# B&R Automation Studio project KeePak_BlissNewScreen
Automation Studio 4.7.5.60 SP

## Configuration MasterConfiguration_ServoRam

### Acp10map.ncm - X20CP0484/Motion/Acp10map.ncm
```
NcMapping (NcSwId=Acp10, DisabledNodesAreHidden=False)
  NcObject 8EI2X2HWT10.xxxx-1a_ncV_AXIS1 (ModuleId=8EI2X2HWT10.xxxx-1a, Type=ncV_AXIS, Channel=1, Disabled=TRUE, ModuleDisabled=FALSE)
  NcObject gServoRam (ModuleId=8EI2X2HWT10.xxxx-1a, Type=ncAXIS, Channel=1, AcoposSimulation=Off, InitParameter=gFeedi, AcoposParameter=brake, Disabled=FALSE, ModuleDisabled=FALSE)
  NcObject 8EI2X2HWT10.xxxx-1_ncV_AXIS1 (ModuleId=8EI2X2HWT10.xxxx-1, Type=ncV_AXIS, Channel=1, Disabled=TRUE, ModuleDisabled=FALSE)
  NcObject gBodyHopper (ModuleId=8EI2X2HWT10.xxxx-1, Type=ncAXIS, Channel=1, AcoposSimulation=Off, InitParameter=gFeedi, AcoposParameter=gBHop, Disabled=FALSE, ModuleDisabled=FALSE)
  NcObject 8EI2X2HWT10.xxxx-1a_ncV_AXIS2 (ModuleId=8EI2X2HWT10.xxxx-1a, Type=ncV_AXIS, Channel=2, Disabled=TRUE, ModuleDisabled=FALSE)
  NcObject gServoPnP (ModuleId=8EI2X2HWT10.xxxx-1a, Type=ncAXIS, Channel=2, AcoposSimulation=Off, InitParameter=gFeedi, AcoposParameter=disablebra, Disabled=FALSE, ModuleDisabled=FALSE)
  NcObject 8EI2X2HWT10.xxxx-1_ncV_AXIS2 (ModuleId=8EI2X2HWT10.xxxx-1, Type=ncV_AXIS, Channel=2, Disabled=TRUE, ModuleDisabled=FALSE)
  NcObject gLeftHopper (ModuleId=8EI2X2HWT10.xxxx-1, Type=ncAXIS, Channel=2, AcoposSimulation=Off, InitParameter=gFeedi, AcoposParameter=gBHop, Disabled=FALSE, ModuleDisabled=FALSE)
  NcObject 8EI2X2HWT10.xxxx-1a_ncV_AXIS3 (ModuleId=8EI2X2HWT10.xxxx-1a, Type=ncV_AXIS, Channel=3, Disabled=TRUE, ModuleDisabled=FALSE)
  NcObject gServoFeed (ModuleId=8EI2X2HWT10.xxxx-1a, Type=ncAXIS, Channel=3, AcoposSimulation=Off, InitParameter=gFeedi, AcoposParameter=disablebra, Disabled=FALSE, ModuleDisabled=FALSE)
  NcObject 8EI2X2HWT10.xxxx-1_ncV_AXIS3 (ModuleId=8EI2X2HWT10.xxxx-1, Type=ncV_AXIS, Channel=3, Disabled=TRUE, ModuleDisabled=FALSE)
  NcObject gRightHopper (ModuleId=8EI2X2HWT10.xxxx-1, Type=ncAXIS, Channel=3, AcoposSimulation=Off, InitParameter=gFeedi, AcoposParameter=gBHop, Disabled=FALSE, ModuleDisabled=FALSE)
```

### BodyHop.mpaxisbasic - X20CP0484/Motion/BodyHop.mpaxisbasic
```
Element mpBodyHopper (Type=mpaxisbasic)
  AxisConfiguration:
    Axis:
      MeasurementUnit = 1
  Alarms = MpAlarmX
    mapp.AlarmX.Core.Configuration:
      [0]:
        Severity = 110
      [1]:
        Severity = 110
      [2]:
        Severity = 110
      [3]:
        Severity = 110
      [4]:
        Severity = 110
      [5]:
        Severity = 110
      [6]:
        Severity = 110
      [7]:
        Severity = 110
      [8]:
        Severity = 110
      [9]:
        Severity = 110
      [10]:
        Severity = 110
      [11]:
        Severity = 110
      [12]:
        Severity = 110
      [13]:
        Severity = 110
      [14]:
        Severity = 110
      [15]:
        Severity = 110
```

### ServoPnP.mpaxisbasic - X20CP0484/Motion/ServoPnP.mpaxisbasic
```
Element mpServoPick (Type=mpaxisbasic)
  AxisConfiguration:
    Axis:
      MeasurementUnit = 1
  Alarms = MpAlarmX
    mapp.AlarmX.Core.Configuration:
      [0]:
        Severity = 110
      [1]:
        Severity = 110
      [2]:
        Severity = 110
      [3]:
        Severity = 110
      [4]:
        Severity = 110
      [5]:
        Severity = 110
      [6]:
        Severity = 110
      [7]:
        Severity = 110
      [8]:
        Severity = 110
      [9]:
        Severity = 110
      [10]:
        Severity = 110
      [11]:
        Severity = 110
      [12]:
        Severity = 110
      [13]:
        Severity = 110
      [14]:
        Severity = 110
      [15]:
        Severity = 110
```

- Safety project (password-protected, skipped)

## Logical view

### Global.var
```iecst
VAR
	GuideCylinder : BOOL;
	gForceBodyKicker : BOOL;
END_VAR
VAR RETAIN
	BodyHopperFirstHomeExecuted : BOOL;
	BodyHopper_EPD : MC_ENDLESS_POSITION;
END_VAR
VAR
	b_ModuleStatus : BOOL;
END_VAR
VAR RETAIN
	CycleCount : UDINT;
END_VAR
VAR
	DistanceAfterLatch : REAL;
	FeedInCycle : BOOL;
	FeedPosFinal : LREAL;
	FeedPositionCapture : LREAL;
	FeedServoBusy : BOOL;
	gActivePage : USINT;
	gAdhesiveCtrlInterface : AdhesiveCtrlInterface_typ;
	gAirPressureAlarmActive : BOOL;
	gAlarmActive : BOOL;
	gAlarmSystemActive : BOOL;
	gAutoTune : BOOL;
	gBodyHopper : ACP10AXIS_typ;
	gBodyHopperInterface : Axis_Interface_typ;
	gBotLinAxis : ACP10AXIS_typ;
	gBotLinAxis_1 : ACP10AXIS_typ;
	gChangePage : USINT;
	gCurrentLimitHit : BOOL;
	gCyclesToFinish : SINT;
	gDownstreamBlocked : BOOL;
END_VAR
VAR RETAIN
	gEndlessPosBot : MC_ENDLESS_POSITION;
	gEndlessPosTop : MC_ENDLESS_POSITION;
END_VAR
VAR
	gFoldPushCtrlInterface : FoldPushCtrlInterface_typ := (Parameters:=(LinMotBotFolder:=(Parameter:=(MpBasicParameters:=(Home:=(Mode:=mpAXIS_HOME_MODE_RESTORE_POS,Position:=0,StartVelocity:=25,HomingVelocity:=5,Acceleration:=500,StartDirection:=mpAXIS_HOME_DIR_NEGATIVE,TorqueLimit:=0.5,BlockDetectionPositionError:=4,PositionErrorStopLimit:=10),Jog:=(Velocity:=2)))),LinMotTopFolder:=(Parameter:=(MpBasicParameters:=(Home:=(Mode:=mpAXIS_HOME_MODE_RESTORE_POS,Position:=0,StartVelocity:=25,HomingVelocity:=5,Acceleration:=500,StartDirection:=mpAXIS_HOME_DIR_NEGATIVE,TorqueLimit:=0.5,BlockDetectionPositionError:=4,PositionErrorStopLimit:=10),Jog:=(Velocity:=2))))));
	gHighSeverityAlarmActive : BOOL;
	gHMI : HMIControl_typ;
	gHomingParameters : Home_Parameters_typ;
	gIO : IO_typ;
	gIsSimulated : BOOL;
	gLeftHopper : ACP10AXIS_typ;
	gLeftHopperInterface : Axis_Interface_typ;
	gLowSeverityAlarmActive : BOOL;
	gModeControlInterface : ModeCtrlInterface_typ;
	gNumActiveAlarms : UDINT;
	gNumAlarms : UDINT;
	gOffDelayCompensation : REAL;
	gOnDelayCompensation : REAL;
	gPassword : ARRAY[0..2] OF STRING[80] := ['','1111','2147'];
	gPnPAtStopPosition : BOOL;
	gPusherOn : BOOL;
	gRamAtStopPosition : BOOL;
	gRamCtrlInterface : RamControlInterface_typ;
	gRamWaitingOnBox : BOOL;
END_VAR
VAR RETAIN
	gRecipeInterface : {REDUND_UNREPLICABLE} RecipeCtrlInterface_typ := (0);
END_VAR
VAR
	gRightHopper : ACP10AXIS_typ;
	gRightHopperInterface : Axis_Interface_typ;
	gSafetyNotOKAlarmActive : BOOL;
	gServoFeed : ACP10AXIS_typ;
	gServoFeedInterface : Axis_Interface_typ;
	gServoFeed_1 : ACP10AXIS_typ;
	gServoPnP : ACP10AXIS_typ;
	gServoPnPInterface : Axis_Interface_typ;
	gServoRam : ACP10AXIS_typ;
	gServoRamInterface : Axis_Interface_typ;
	gServoRam_1 : ACP10AXIS_typ;
	gSoftwareReset : BOOL;
	gTopLinAxis : ACP10AXIS_typ;
	gTopLinAxis_1 : ACP10AXIS_typ;
	gUserLevel : USINT;
	gVacCtrlInterface : VacCtrlInterface_typ;
	HoperLowStop : BOOL;
	HopperLowTime : TIME := T#7s;
	InfeedBoxPresent : BOOL;
END_VAR
VAR RETAIN
	LeftHopperFirstHomeExecuted : BOOL;
	LeftHopper_EPD : MC_ENDLESS_POSITION;
	LubeCount : UDINT;
END_VAR
VAR
	LubricationOK : BOOL;
	Melter : DUT_NDSN_Flex;
	PhotoEyeSeen : BOOL;
END_VAR
VAR RETAIN
	RightHopperFirstHomeExecuted : BOOL;
	RightHopper_EPD : MC_ENDLESS_POSITION;
	ServoFeedFirstHomeExecuted : BOOL;
	ServoFeed_EPD : MC_ENDLESS_POSITION;
END_VAR
VAR
	ServoPnPAutoHome : BOOL;
END_VAR
VAR RETAIN
	ServoPnPFirstHomeExecuted : BOOL;
	ServoPnP_EPD : MC_ENDLESS_POSITION;
END_VAR
VAR
	ServoRamAutoHome : BOOL;
	ServoRamBusy : BOOL;
	ServoRamClear : BOOL;
END_VAR
VAR RETAIN
	ServoRamFirstHomeExecuted : BOOL;
END_VAR
VAR
	ServoRamTrigger : BOOL;
END_VAR
VAR RETAIN
	ServoRam_EPD : MC_ENDLESS_POSITION;
END_VAR
VAR
	StopFeed : BOOL;
END_VAR
```

### Program Logical/Actuators/NordsonComm/NordsonMBComm

#### MbApp.st
```iecst
(********************************************************************
 * COPYRIGHT -- Bernecker + Rainer
 ********************************************************************
 * Program: MbApp
 * File: MbApp.st
 * Author: Bernecker + Rainer
 * Created: October 22, 2009
 ********************************************************************
 * Implementation of program MbApp
 * State Nomenclature: "request" is a write to the nordson melter asking for some data
 * 					   "read" is a read from the nordson melter of the previously requested data
 *                     "write" is a write to the nordson melter asking to write some data to the melter
 *                     "verify" is a read from the nordson melter where we check to see that the write was accepted
 ********************************************************************)

PROGRAM _INIT

	NordsonTxPacket.Byte0_MelterControl := 16#1;
	NordsonTxPacket.Byte1_Command := 3;
	NordsonTxPacket.Byte2_Data_Index := 16#78;
	NordsonTxPacket.Byte3_Channel_Num := 16#3;
	NordsonTxPacket.Byte4_5_WriteData := 0;
	NordsonTxPacket.Byte6_7_Mot1Spd := 0;
	NordsonTxPacket.Byte8_9_Mot2Spd := 0;
	NordsonTxPacket.Byte10_11_Mot3Spd := 0;
	NordsonTxPacket.Byte12_13_Mot4Spd := 0;
	NordsonTxPacket.Byte14_15_NotUsed := 0;

	state := MB_IDLE;

	(* init values *)
	mb_station 			:= 'IF2.ST2';					(* path to modbus station *)
	write_register_address	:= 1024;						(* register address on modbus station *)
	read_register_address	:= 0;						(* register address on modbus station *)
	num_registers_to_write := 8;
	num_registers_to_read := 8;

	testChannel := CHANNEL_ACT_TEMP_START;
	testIdx := IDX_ACT_TEMP;

	gAdhesiveCtrlInterface.Commands.MelterOn := TRUE;
	gAdhesiveCtrlInterface.Commands.PumpsOn := TRUE;
	//gAdhesiveCtrlInterface.Parameters.NordsonComms.StandbyTimeoutTime := T#2h;
	//Removed Standby due to Waco machine going into Standby at random times. Added 05/15/2024

	FirstTimeCopySetTemps := FALSE;

END_PROGRAM

PROGRAM _CYCLIC

	IF(gAdhesiveCtrlInterface.Parameters.FeedbackIsModbusTCP) THEN
		gHMI.StatusDatapoints.NordsonModbusSDP := UNHIDE + UNLOCK;
	ELSE
		gHMI.StatusDatapoints.NordsonModbusSDP := HIDE + LOCK;
	END_IF

	StandbyTimer.IN := NOT(gRamCtrlInterface.Status.Running) AND NOT(gAdhesiveCtrlInterface.Commands.MelterStandbyOn);
	StandbyTimer.PT := gAdhesiveCtrlInterface.Parameters.NordsonComms.StandbyTimeoutTime;
	StandbyTimer();

	IF(StandbyTimer.Q) THEN
		gAdhesiveCtrlInterface.Commands.MelterStandbyOn := TRUE;
	END_IF

	//clearing standby on command shiuld turn standby off. Changed standbyoff to True
	IF(gAdhesiveCtrlInterface.Commands.MelterStandbyOff) THEN
		gAdhesiveCtrlInterface.Commands.MelterStandbyOff := TRUE;
		gAdhesiveCtrlInterface.Commands.MelterStandbyOn := FALSE;
	END_IF

	IF((gAdhesiveCtrlInterface.Status.NordsonInStandby) AND (gAdhesiveCtrlInterface.Parameters.FeedbackIsModbusTCP)) THEN
		gHMI.StatusDatapoints.NordsonStandbyOffSDP := UNHIDE + UNLOCK;
	ELSE
		gHMI.StatusDatapoints.NordsonStandbyOffSDP := HIDE + LOCK;
	END_IF

	//if nordson feedback is bypassed, the error count should reset to 0
	IF gAdhesiveCtrlInterface.Parameters.NordsonComms.ByPassFeedback THEN
		gAdhesiveCtrlInterface.Parameters.NordsonComms.ConsecutiveErrorCount := 0;
	END_IF

	CASE state OF

		MB_IDLE:
			FeedbackCycleTimer.IN := ((gAdhesiveCtrlInterface.Parameters.FeedbackIsModbusTCP) AND (gAdhesiveCtrlInterface.Parameters.NordsonComms.ByPassFeedback = FALSE));

			IF(gAdhesiveCtrlInterface.Parameters.FeedbackIsModbusTCP = FALSE) THEN
				gAdhesiveCtrlInterface.Parameters.NordsonComms.ConsecutiveErrorCount := 0;
			END_IF

			IF(gAdhesiveCtrlInterface.Commands.WriteChannelTemp) THEN
				gAdhesiveCtrlInterface.Commands.WriteChannelTemp := FALSE;
				TempChannelToWrite := 0;
				state := MB_WRITE_SET_TEMP;

			ELSIF(FeedbackCycleTimer.Q) THEN
				FeedbackCycleTimer.IN := FALSE;
				state := MB_REQUEST_MELTER_STATUS;
			END_IF

		MB_REQUEST_MELTER_STATUS:

			WriteMultipleRegisters.enable := 1;
			NordsonTxPacket.Byte0_MelterControl := MelterCmd;
			NordsonTxPacket.Byte1_Command := READ_COMMAND;
			NordsonTxPacket.Byte2_Data_Index := IDX_MELTER_STATUS;
			NordsonTxPacket.Byte3_Channel_Num := 0;

			IF((WriteMultipleRegisters.status = ERR_FUB_ENABLE_FALSE) OR (WriteMultipleRegisters.status = ERR_FUB_BUSY)) THEN
				//do nothing
			ELSIF(WriteMultipleRegisters.status = ERR_OK) THEN
				WriteMultipleRegisters.enable := 0;
				state := MB_READ_MELTER_STATUS;
			ELSE
				WriteMultipleRegisters.enable := 0;
				MBError := WriteMultipleRegisters.status;
				state := MB_ERROR;
			END_IF

		MB_READ_MELTER_STATUS:

			ReadMultipleRegisters.enable := 1;

			IF((ReadMultipleRegisters.status = ERR_FUB_ENABLE_FALSE) OR (ReadMultipleRegisters.status = ERR_FUB_BUSY)) THEN
				//do nothing
			ELSIF(ReadMultipleRegisters.status = ERR_OK) THEN

				ReadMultipleRegisters.enable := 0;

				IF(NordsonRxPacket.Byte2_Ack_Data_Index = NordsonTxPacket.Byte2_Data_Index) THEN

					gAdhesiveCtrlInterface.Parameters.NordsonComms.MelterStatus := NordsonRxPacket.Byte4_5_Read_Data_0;
					gAdhesiveCtrlInterface.Parameters.NordsonComms.MelterIsOn := (gAdhesiveCtrlInterface.Parameters.NordsonComms.MelterStatus <> 8); //melter status == 8 => melter is not on

					DecodeStatus;

					//the melter MUST see a 0 for its ON command before it sees a 1. Send a 0 if the unit is faulted OR we have previously told it to turn on. and it never came on
				//	IF((gAdhesiveCtrlInterface.Parameters.NordsonComms.UnitFaulted) OR ((gAdhesiveCtrlInterface.Parameters.NordsonComms.MelterIsOn = FALSE) AND (NordsonTxPacket.Byte0_MelterControl.0 = TRUE))) THEN
					IF((gAdhesiveCtrlInterface.Parameters.NordsonComms.MelterIsOn = FALSE) AND (NordsonTxPacket.Byte0_MelterControl.0 = TRUE)) THEN
						MelterCmd := MELTER_OFF + PUMPS_OFF; //melter off, pumps off
					ELSE

						MelterCmd := 0;
						IF(gAdhesiveCtrlInterface.Commands.MelterOn) THEN
							MelterCmd := MelterCmd + MELTER_ON;
						END_IF

						IF((gAdhesiveCtrlInterface.Commands.PumpsOn) AND (gAdhesiveCtrlInterface.Status.UnitReady)) THEN
							MelterCmd := MelterCmd + PUMPS_ON; //only turn the pump on if the melter is ready
						END_IF

						IF((gAdhesiveCtrlInterface.Commands.MelterStandbyOn = FALSE) OR ((gAdhesiveCtrlInterface.Status.NordsonInStandby = FALSE) AND NordsonTxPacket.Byte0_MelterControl.6 = TRUE)) THEN
							//do not standby on
						ELSIF (gAdhesiveCtrlInterface.Commands.MelterStandbyOn = TRUE) THEN
							MelterCmd := MelterCmd + STANDBY_ON; //only turn the pump on if the melter is ready
						END_IF
					END_IF

					state := MB_REQUEST_SET_TEMPS;
				ELSE
					//stay in this state and re-execute read
				END_IF

			ELSE
				ReadMultipleRegisters.enable := 0;
				MBError := ReadMultipleRegisters.status;
				state := MB_ERROR;
			END_IF

		MB_REQUEST_SET_TEMPS:

			WriteMultipleRegisters.enable := 1;
			NordsonTxPacket.Byte0_MelterControl := MelterCmd;
			NordsonTxPacket.Byte1_Command := READ_COMMAND;
			NordsonTxPacket.Byte2_Data_Index := IDX_SET_TEMP;
			NordsonTxPacket.Byte3_Channel_Num := CHANNEL_SET_TEMP_START;

			IF((WriteMultipleRegisters.status = ERR_FUB_ENABLE_FALSE) OR (WriteMultipleRegisters.status = ERR_FUB_BUSY)) THEN
				//do nothing
			ELSIF(WriteMultipleRegisters.status = ERR_OK) THEN
				WriteMultipleRegisters.enable := 0;
				gAdhesiveCtrlInterface.Parameters.NordsonComms.ConsecutiveErrorCount := 0;
				state := MB_READ_SET_TEMPS;
			ELSE
				WriteMultipleRegisters.enable := 0;
				MBError := WriteMultipleRegisters.status;
				state := MB_ERROR;
			END_IF

		MB_READ_SET_TEMPS:

			ReadMultipleRegisters.enable := 1;

			IF((ReadMultipleRegisters.status = ERR_FUB_ENABLE_FALSE) OR (ReadMultipleRegisters.status = ERR_FUB_BUSY)) THEN
				//do nothing
			ELSIF(ReadMultipleRegisters.status = ERR_OK) THEN
				ReadMultipleRegisters.enable := 0;
				gAdhesiveCtrlInterface.Parameters.NordsonComms.ConsecutiveErrorCount := 0;

				IF((NordsonRxPacket.Byte2_Ack_Data_Index = NordsonTxPacket.Byte2_Data_Index) AND
					(NordsonRxPacket.Byte3_Ack_Channel_Num = NordsonTxPacket.Byte3_Channel_Num)) THEN

					DecodeStatus;

					gAdhesiveCtrlInterface.Parameters.NordsonComms.ChannelSetTempActual[0] := NordsonRxPacket.Byte4_5_Read_Data_0;
					gAdhesiveCtrlInterface.Parameters.NordsonComms.ChannelSetTempActual[1] := NordsonRxPacket.Byte6_7_Read_Data_1;
					gAdhesiveCtrlInterface.Parameters.NordsonComms.ChannelSetTempActual[2] := NordsonRxPacket.Byte8_9_Read_Data_2;
					gAdhesiveCtrlInterface.Parameters.NordsonComms.ChannelSetTempActual[3] := NordsonRxPacket.Byte10_11_Read_Data_3;
					gAdhesiveCtrlInterface.Parameters.NordsonComms.ChannelSetTempActual[4] := NordsonRxPacket.Byte12_13_Read_Data_4;
                    gAdhesiveCtrlInterface.Parameters.NordsonComms.ChannelSetTempActual[5] := NordsonRxPacket.Byte14_15_Read_Data_5;
//                    gAdhesiveCtrlInterface.Parameters.NordsonComms.ChannelSetTempActual[6] := NordsonRxPacket.Byte16_17_Read_Data_6;
//                    gAdhesiveCtrlInterface.Parameters.NordsonComms.ChannelSetTempActual[7] := NordsonRxPacket.Byte18_19_Read_Data_7;

                    IF (FirstTimeCopySetTemps = FALSE) THEN
						gAdhesiveCtrlInterface.Parameters.NordsonComms.ChannelSetTempRequested := gAdhesiveCtrlInterface.Parameters.NordsonComms.ChannelSetTempActual;
						FirstTimeCopySetTemps := TRUE;
					END_IF

					state := MB_REQUEST_ACT_TEMPS; //for now, just go back to idle. Future versions need to read more stuff
				ELSE
					//stay in this state and re-execute read
				END_IF
			ELSE
				ReadMultipleRegisters.enable := 0;
				MBError := ReadMultipleRegisters.status;
				state := MB_ERROR;
			END_IF

		MB_REQUEST_ACT_TEMPS:

			WriteMultipleRegisters.enable := 1;
			NordsonTxPacket.Byte0_MelterControl := MelterCmd;
			NordsonTxPacket.Byte1_Command := READ_COMMAND;
			NordsonTxPacket.Byte2_Data_Index := IDX_ACT_TEMP;
			NordsonTxPacket.Byte3_Channel_Num := CHANNEL_ACT_TEMP_START;

			IF((WriteMultipleRegisters.status = ERR_FUB_ENABLE_FALSE) OR (WriteMultipleRegisters.status = ERR_FUB_BUSY)) THEN
				//do nothing
			ELSIF(WriteMultipleRegisters.status = ERR_OK) THEN
				WriteMultipleRegisters.enable := 0;
				state := MB_READ_ACT_TEMPS;
			ELSE
				WriteMultipleRegisters.enable := 0;
				MBError := WriteMultipleRegisters.status;
				state := MB_ERROR;
			END_IF

		MB_READ_ACT_TEMPS:

			ReadMultipleRegisters.enable := 1;

			IF((ReadMultipleRegisters.status = ERR_FUB_ENABLE_FALSE) OR (ReadMultipleRegisters.status = ERR_FUB_BUSY)) THEN
				//do nothing
			ELSIF(ReadMultipleRegisters.status = ERR_OK) THEN
				ReadMultipleRegisters.enable := 0;

				IF((NordsonRxPacket.Byte2_Ack_Data_Index = NordsonTxPacket.Byte2_Data_Index) AND
					(NordsonRxPacket.Byte3_Ack_Channel_Num = NordsonTxPacket.Byte3_Channel_Num)) THEN

					DecodeStatus;

					gAdhesiveCtrlInterface.Parameters.NordsonComms.ChannelActTemp[0] := NordsonRxPacket.Byte4_5_Read_Data_0;
					gAdhesiveCtrlInterface.Parameters.NordsonComms.ChannelActTemp[1] := NordsonRxPacket.Byte6_7_Read_Data_1;
					gAdhesiveCtrlInterface.Parameters.NordsonComms.ChannelActTemp[2] := NordsonRxPacket.Byte8_9_Read_Data_2;
					gAdhesiveCtrlInterface.Parameters.NordsonComms.ChannelActTemp[3] := NordsonRxPacket.Byte10_11_Read_Data_3;
					gAdhesiveCtrlInterface.Parameters.NordsonComms.ChannelActTemp[4] := NordsonRxPacket.Byte12_13_Read_Data_4;
                    gAdhesiveCtrlInterface.Parameters.NordsonComms.ChannelActTemp[5] := NordsonRxPacket.Byte14_15_Read_Data_5;
//                    gAdhesiveCtrlInterface.Parameters.NordsonComms.ChannelActTemp[6] := NordsonRxPacket.Byte16_17_Read_Data_6;
//                    gAdhesiveCtrlInterface.Parameters.NordsonComms.ChannelActTemp[7] := NordsonRxPacket.Byte18_19_Read_Data_7;
//                    gAdhesiveCtrlInterface.Parameters.NordsonComms.ChannelActTemp[8] := NordsonRxPacket.Byte20_21_Read_Data_8;
//                    gAdhesiveCtrlInterface.Parameters.NordsonComms.ChannelActTemp[9] := NordsonRxPacket.Byte22_23_Read_Data_9;
//                    gAdhesiveCtrlInterface.Parameters.NordsonComms.ChannelActTemp[10] := NordsonRxPacket.Byte24_25_Read_Data_10;

					state := MB_REQUEST_ATS_ALARMS;
				ELSE
					//stay in this state and re-execute read
				END_IF

			ELSE
				ReadMultipleRegisters.enable := 0;
				MBError := ReadMultipleRegisters.status;
				state := MB_ERROR;
			END_IF

		MB_REQUEST_ATS_ALARMS:

			WriteMultipleRegisters.enable := 1;
			NordsonTxPacket.Byte0_MelterControl := MelterCmd;
			NordsonTxPacket.Byte1_Command := READ_COMMAND;
			NordsonTxPacket.Byte2_Data_Index := IDX_ATS_ALARMS;

			IF((WriteMultipleRegisters.status = ERR_FUB_ENABLE_FALSE) OR (WriteMultipleRegisters.status = ERR_FUB_BUSY)) THEN
				//do nothing
			ELSIF(WriteMultipleRegisters.status = ERR_OK) THEN
				WriteMultipleRegisters.enable := 0;
				state := MB_READ_ATS_ALARMS;
			ELSE
				WriteMultipleRegisters.enable := 0;
				MBError := WriteMultipleRegisters.status;
				state := MB_ERROR;
			END_IF

		MB_READ_ATS_ALARMS:

			ReadMultipleRegisters.enable := 1;

			IF((ReadMultipleRegisters.status = ERR_FUB_ENABLE_FALSE) OR (ReadMultipleRegisters.status = ERR_FUB_BUSY)) THEN
				//do nothing
			ELSIF(ReadMultipleRegisters.status = ERR_OK) THEN
				ReadMultipleRegisters.enable := 0;

				IF(NordsonRxPacket.Byte2_Ack_Data_Index = NordsonTxPacket.Byte2_Data_Index) THEN

					DecodeStatus;

					gAdhesiveCtrlInterface.Status.ATS_AddOnOverLimit := NordsonRxPacket.Byte4_5_Read_Data_0.0;
					gAdhesiveCtrlInterface.Status.ATS_AddOnUnderLimit := NordsonRxPacket.Byte4_5_Read_Data_0.1;

					state := MB_IDLE;
				ELSE
					//stay in this state and re-execute read
				END_IF

			ELSE
				ReadMultipleRegisters.enable := 0;
				MBError := ReadMultipleRegisters.status;
				state := MB_ERROR;
			END_IF

		MB_WRITE_SET_TEMP:

			WriteMultipleRegisters.enable := 1;
			NordsonTxPacket.Byte0_MelterControl := MelterCmd;
			NordsonTxPacket.Byte1_Command := WRITE_COMMAND;
			NordsonTxPacket.Byte2_Data_Index := IDX_SET_TEMP;
			NordsonTxPacket.Byte3_Channel_Num := TempChannelToWrite + 1; //TempChannelToWrite starts counting at 0, but nordson melter starts counting at 1
			NordsonTxPacket.Byte4_5_WriteData := gAdhesiveCtrlInterface.Parameters.NordsonComms.ChannelSetTempRequested[TempChannelToWrite];

			IF((WriteMultipleRegisters.status = ERR_FUB_ENABLE_FALSE) OR (WriteMultipleRegisters.status = ERR_FUB_BUSY)) THEN
				//do nothing
			ELSIF(WriteMultipleRegisters.status = ERR_OK) THEN
				WriteMultipleRegisters.enable := 0;
				state := MB_VERIFY_SET_TEMP_WRITE;
			ELSE
				WriteMultipleRegisters.enable := 0;
				MBError := WriteMultipleRegisters.status;
				state := MB_ERROR;
			END_IF

		MB_VERIFY_SET_TEMP_WRITE:

			ReadMultipleRegisters.enable := 1;

			IF((ReadMultipleRegisters.status = ERR_FUB_ENABLE_FALSE) OR (ReadMultipleRegisters.status = ERR_FUB_BUSY)) THEN
				//do nothing
			ELSIF(ReadMultipleRegisters.status = ERR_OK) THEN
				ReadMultipleRegisters.enable := 0;

				IF((NordsonRxPacket.Byte2_Ack_Data_Index = NordsonTxPacket.Byte2_Data_Index) AND
					(NordsonRxPacket.Byte3_Ack_Channel_Num = NordsonTxPacket.Byte3_Channel_Num)) THEN

					DecodeStatus;

					IF(TempChannelToWrite < NUM_NORDSON_TEMP_ZONES_M1) THEN
						IF(TempChannelToWrite = 0) THEN
							TempChannelToWrite := 2; //channel 0 and 1 get the same temp, no need to re-write channel 1
							state := MB_WRITE_SET_TEMP;
						ELSE
							TempChannelToWrite := TempChannelToWrite + 1; //set the temperature for the next channel (Skip channel 2). Machine has 3 total channels
							state := MB_WRITE_SET_TEMP;
						END_IF
					ELSE
						state := MB_IDLE;
					END_IF
				ELSE
					//stay in this state and re-execute read
				END_IF

			ELSE
				ReadMultipleRegisters.enable := 0;
				MBError := ReadMultipleRegisters.status;
				state := MB_ERROR;
			END_IF

		MB_REQUEST_ADH_USE:

			WriteMultipleRegisters.enable := 1;
			NordsonTxPacket.Byte0_MelterControl := MelterCmd;
			NordsonTxPacket.Byte1_Command := READ_COMMAND;
			NordsonTxPacket.Byte2_Data_Index := IDX_ADHESIVE_HOUR;
			NordsonTxPacket.Byte3_Channel_Num := CHANNEL_ADHESIVE_HOUR;

			IF((WriteMultipleRegisters.status = ERR_FUB_ENABLE_FALSE) OR (WriteMultipleRegisters.status = ERR_FUB_BUSY)) THEN
				//do nothing
			ELSIF(WriteMultipleRegisters.status = ERR_OK) THEN
				WriteMultipleRegisters.enable := 0;
				state := MB_READ_ACT_TEMPS;
			ELSE
				WriteMultipleRegisters.enable := 0;
				MBError := WriteMultipleRegisters.status;
				state := MB_ERROR;
			END_IF

		MB_READ_ADH_USE:

			ReadMultipleRegisters.enable := 1;

			IF((ReadMultipleRegisters.status = ERR_FUB_ENABLE_FALSE) OR (ReadMultipleRegisters.status = ERR_FUB_BUSY)) THEN
				//do nothing
			ELSIF(ReadMultipleRegisters.status = ERR_OK) THEN
				ReadMultipleRegisters.enable := 0;

				IF((NordsonRxPacket.Byte2_Ack_Data_Index = NordsonTxPacket.Byte2_Data_Index) AND
					(NordsonRxPacket.Byte3_Ack_Channel_Num = NordsonTxPacket.Byte3_Channel_Num)) THEN

					//	NordsonData.AdhesiveUsePerHour := NordsonRxPacket.Byte4_5_Read_Data_0 + (NordsonRxPacket.Byte6_7_Read_Data_1*(65536)); //data 0 + data 1 shifted up 16 bits

					state := MB_READ_ACT_TEMPS;
				ELSE
					//stay in this state and re-execute read
				END_IF
			END_IF

		MB_WRITE_REGISTERS:

			WriteMultipleRegisters.enable := 1;
			NordsonTxPacket.Byte0_MelterControl := MELTER_ON;
			NordsonTxPacket.Byte1_Command := READ_COMMAND;
			NordsonTxPacket.Byte2_Data_Index := testChannel;
			NordsonTxPacket.Byte3_Channel_Num := testIdx;

			IF((WriteMultipleRegisters.status = ERR_FUB_ENABLE_FALSE) OR (WriteMultipleRegisters.status = ERR_FUB_BUSY)) THEN
				//do nothing
			ELSIF(WriteMultipleRegisters.status = ERR_OK) THEN
				WriteMultipleRegisters.enable := 0;
				state := MB_READ_ACT_TEMPS;
			ELSE
				WriteMultipleRegisters.enable := 0;
				MBError := WriteMultipleRegisters.status;
				state := MB_ERROR;
			END_IF

		MB_READ_REGISTERS:

			ReadMultipleRegisters.enable := 1;

			IF((ReadMultipleRegisters.status = ERR_FUB_ENABLE_FALSE) OR (ReadMultipleRegisters.status = ERR_FUB_BUSY)) THEN
				//do nothing
			ELSIF(ReadMultipleRegisters.status = ERR_OK) THEN
				ReadMultipleRegisters.enable := 0;
				state := MB_IDLE;
			ELSE
				ReadMultipleRegisters.enable := 0;
				MBError := ReadMultipleRegisters.status;
				state := MB_ERROR;
			END_IF

		MB_ERROR:
			gAdhesiveCtrlInterface.Parameters.NordsonComms.ConsecutiveErrorCount := gAdhesiveCtrlInterface.Parameters.NordsonComms.ConsecutiveErrorCount + 1;
		state := MB_IDLE; //keep re-trying indefinetly, logic below will set/reset alarms alarm

	END_CASE;

	IF EDGEPOS(gAdhesiveCtrlInterface.Parameters.NordsonComms.ConsecutiveErrorCount >= 10) THEN
		MpAlarmXSet(gAlarmXCore, ALARM_NORDSON_COMMS);
	ELSIF EDGENEG(gAdhesiveCtrlInterface.Parameters.NordsonComms.ConsecutiveErrorCount >= 10)THEN
		MpAlarmXReset(gAlarmXCore, ALARM_NORDSON_COMMS);
	END_IF

	IF EDGEPOS(gAdhesiveCtrlInterface.Status.ATS_AddOnOverLimit) THEN
		MpAlarmXSet(gAlarmXCore, ALARM_ATS_OVERLIMIT);
	ELSIF EDGENEG(gAdhesiveCtrlInterface.Status.ATS_AddOnOverLimit)THEN
		MpAlarmXReset(gAlarmXCore, ALARM_ATS_OVERLIMIT);
	END_IF

	IF EDGEPOS(gAdhesiveCtrlInterface.Status.ATS_AddOnUnderLimit) THEN
		MpAlarmXSet(gAlarmXCore, ALARM_ATS_UNDERLIMIT);
	ELSIF EDGENEG(gAdhesiveCtrlInterface.Status.ATS_AddOnUnderLimit)THEN
		MpAlarmXReset(gAlarmXCore, ALARM_ATS_UNDERLIMIT);
	END_IF

	IF EDGEPOS(gAdhesiveCtrlInterface.Status.NordsonInStandby) THEN
		MpAlarmXSet(gAlarmXCore, ALARM_NORDSON_STANDBY);
	ELSIF EDGENEG(gAdhesiveCtrlInterface.Status.NordsonInStandby)THEN
		MpAlarmXReset(gAlarmXCore, ALARM_NORDSON_STANDBY);
	END_IF

	//force unit ready and unit faulted status flags if ModbusTCP control is selected and bypass is enabled
	IF(gAdhesiveCtrlInterface.Parameters.FeedbackIsModbusTCP AND gAdhesiveCtrlInterface.Parameters.NordsonComms.ByPassFeedback) THEN
		gAdhesiveCtrlInterface.Parameters.NordsonComms.UnitReady := TRUE;
		gAdhesiveCtrlInterface.Parameters.NordsonComms.UnitFaulted := FALSE;
		gAdhesiveCtrlInterface.Status.ATS_AddOnOverLimit := FALSE;
		gAdhesiveCtrlInterface.Status.ATS_AddOnUnderLimit := FALSE;
	END_IF

	//Must be called after state machine. Do not move any function calls that are already below this line
	WriteMultipleRegisters.pStation := ADR(mb_station);
	WriteMultipleRegisters.startAddress := write_register_address;
	WriteMultipleRegisters.nrRegisters := num_registers_to_write;
	WriteMultipleRegisters.pData := ADR(NordsonTxPacket);
	WriteMultipleRegisters.dataSize := SIZEOF(NordsonTxPacket);
	WriteMultipleRegisters();

	ReadMultipleRegisters.pStation := ADR(mb_station);
	ReadMultipleRegisters.startAddress := read_register_address;
	ReadMultipleRegisters.nrRegisters := num_registers_to_read;
	ReadMultipleRegisters.pData := ADR(NordsonRxPacket);
	ReadMultipleRegisters.dataSize := SIZEOF(NordsonRxPacket);
	ReadMultipleRegisters();

	FeedbackCycleTimer.PT := gAdhesiveCtrlInterface.Parameters.NordsonComms.FeedbackTime;
	FeedbackCycleTimer();

				END_PROGRAM
```

### Program Logical/AsSafetySolution/SafetySample

#### SafetySample.st
```iecst
(********************************************************************
 * COPYRIGHT -- Bernecker + Rainer
 ********************************************************************
 * Program: SafetySample
 * File: SafetySample.st
 * Author: B&R
 ********************************************************************
 * Implementation of program SafetySample
 ********************************************************************)

PROGRAM _INIT

(*KEEPAK specific hard coded values *)
	remotecmd.Password 			:= 'safety';				(* password *)
	remotecmd.NewPassword	 	:= 'safety';				(* password *)
	appcmd1.Password 			:= 'safety';
	datacmd1.Password 			:= 'safety';
	datacmd2.Password 			:= 'safety';

	visuUsedSLIDRemote			:= 1;
	visuUsedSLIDData			:= 1;

	slxused						:= 1;
	Station						:= 'IF6.ST6';
	visuEnableMachineOptions	:= 1;
	visuEnableModuleFlags		:= 1;

	visuLockSDP					:= 2;

(* command structure for remote control FUB *)
remotecmd.Version := safeVERSION_R107;	(* version *)
//remotecmd.Password := '';				(* password *)

(* command structure for application download *)
appcmd1.Version := safeVERSION_R107;	(* version *)
//appcmd1.Password := '';					(* password *)
appcmd1.ApplicationID := 1;				(* application id *)

(* command structure for machine options download *)
datacmd1.Version := safeVERSION_R107;								(* version *)
//datacmd1.Password := '';											(* password *)
datacmd1.pDeviceListInput := ADR(visuDeviceListInput);				(* device list *)
datacmd1.pMachineOptionsInput := ADR(dataMachineOptionsBitInput);	(* bit machine options *)
datacmd1.pModuleFlagsInput := ADR(dataModuleFlagsInput);			(* module flags *)
datacmd1.pAcknMachineOptions := ADR(dataAcknMachineOptions);		(* acknowledge information *)

(* command structure for extended machine options *)
datacmd2.Version := safeVERSION_R107;					(* version *)
//datacmd2.Password := '';								(* password *)
datacmd2.pIntDataInput := ADR(visuIntInput);			(* INT channels *)
datacmd2.NumberIntInput := 1;							(* number of INT channels *)
datacmd2.pUintDataInput := ADR(visuUintInput);			(* UINT channels *)
datacmd2.NumberUintInput := 1;							(* number of UINT channels *)
datacmd2.pDintDataInput := ADR(visuDintInput);			(* DINT channels *)
datacmd2.NumberDintInput := 1;							(* number of DINT channels *)
datacmd2.pUdintDataInput := ADR(visuUdintInput);		(* UDINT channels *)
datacmd2.NumberUdintInput := 1;							(* number of UDINT channels *)
datacmd2.pAcknMachineOptions := ADR(visuAcknExtData);	(* acknowledge information *)

(* hide elements in visualization *)
FOR xcnt := 0 TO SIZEOF(statusButtonActiv) - 1 DO
	statusButtonActiv[xcnt] := 1;
END_FOR

(* hide elements in visualization *)
statusButtonUnlockApp := 1;
statusButtonUnlockData := 1;
statusAcknInfoData := 1;
statusButtonUnlockExtData := 1;
statusAcknInfoExtData := 1;
statusDialog := 1;

(* set SafeLOGIC ID *)
visuUsedSLIDRemote := 1;
visuUsedSLIDData := 1;

END_PROGRAM

PROGRAM _CYCLIC
	(****************************************************************************************************************************************)
	(****************************************************************************************************************************************)
	(****************************************************************************************************************************************)
	(* show dialog to ackn command *)
	IF (dialogRemoteCmd = 1) THEN
		statusDialog := 0;
		dialogRemoteCmd := 0;
		indexButtonLeft := 0;
		indexButtonRight := 1;
		indexHeaderText := 0;
		IF (remotecmd.Data = safeCMD_SK_FORMAT) THEN
			indexMessageText := 0;
		ELSIF (remotecmd.Data = safeCMD_SK_XCHG) THEN
			indexMessageText := 1;
		ELSIF (remotecmd.Data = safeCMD_1_UDID_ACKN) THEN
			indexMessageText := 2;
		ELSIF (remotecmd.Data = safeCMD_2_UDID_ACKN) THEN
			indexMessageText := 3;
		ELSIF (remotecmd.Data = safeCMD_3_UDID_ACKN) THEN
			indexMessageText := 4;
		ELSIF (remotecmd.Data = safeCMD_4_UDID_ACKN) THEN
			indexMessageText := 5;
		ELSIF (remotecmd.Data =  safeCMD_N_UDID_ACKN) THEN
			indexMessageText := 6;
		ELSIF (remotecmd.Data =  safeCMD_CLEAR_DATA) THEN
			indexMessageText := 7;
		ELSIF (remotecmd.Data = safeCMD_FW_ACKN) THEN
			indexMessageText := 8;
		ELSIF (remotecmd.Data = safeCMD_RESET) THEN
			indexMessageText := 9;
		END_IF
	END_IF

	(* if dialog is ackn execute fub *)
	IF (dialogButtonLeft = 1 AND indexHeaderText = 0) THEN
		executeRemoteCmd := 1;
		dialogButtonLeft := 0;
		statusDialog := 1;
	ELSIF (dialogButtonRight = 1 AND indexHeaderText = 0) THEN
		dialogButtonRight := 0;
		statusDialog := 1;
	END_IF

	(* password must be at least 6 characters long *)
	IF brsstrlen(ADR(remotecmd.NewPassword)) < 6 THEN
		statusSetPassword := 2;
	ELSE
		statusSetPassword := 0;
	END_IF

	safeRemoteControl_0(SafeLOGICID := visuUsedSLIDRemote, Execute := executeRemoteCmd, pCommandData := ADR(remotecmd));
	(* reset execution flag *)
	IF (safeRemoteControl_0.Done = 1 OR safeRemoteControl_0.Error = 1) THEN
		executeRemoteCmd := 0;
	END_IF

	(* variables for visualization *)
	IF (safeRemoteControl_0.SafeLOGICStatus.SafeKEYChanged = 1) THEN
		FOR xcnt := 0 TO SIZEOF(statusButtonActiv) - 1 DO
			statusButtonActiv[xcnt] := 1;
 			statusButtonInactiv[xcnt] := 0;
		END_FOR
		statusButtonActiv[1] := 0;
 		statusButtonInactiv[1] := 1;
	ELSIF (safeRemoteControl_0.SafeLOGICStatus.NumberOfUDIDMismatches = 1 AND safeRemoteControl_0.SafeLOGICStatus.Scanning = 0) THEN
		FOR xcnt := 0 TO SIZEOF(statusButtonActiv) - 1 DO
			statusButtonActiv[xcnt] := 1;
 			statusButtonInactiv[xcnt] := 0;
		END_FOR
		statusButtonActiv[3] := 0;
 		statusButtonInactiv[3] := 1;
	ELSIF (safeRemoteControl_0.SafeLOGICStatus.NumberOfUDIDMismatches = 2 AND safeRemoteControl_0.SafeLOGICStatus.Scanning = 0) THEN
		FOR xcnt := 0 TO SIZEOF(statusButtonActiv) - 1 DO
			statusButtonActiv[xcnt] := 1;
 			statusButtonInactiv[xcnt] := 0;
		END_FOR
		statusButtonActiv[4] := 0;
 		statusButtonInactiv[4] := 1;
	ELSIF (safeRemoteControl_0.SafeLOGICStatus.NumberOfUDIDMismatches = 3 AND safeRemoteControl_0.SafeLOGICStatus.Scanning = 0) THEN
		FOR xcnt := 0 TO SIZEOF(statusButtonActiv) - 1 DO
			statusButtonActiv[xcnt] := 1;
 			statusButtonInactiv[xcnt] := 0;
		END_FOR
		statusButtonActiv[5] := 0;
 		statusButtonInactiv[5] := 1;
	ELSIF (safeRemoteControl_0.SafeLOGICStatus.NumberOfUDIDMismatches = 4 AND safeRemoteControl_0.SafeLOGICStatus.Scanning = 0) THEN
		FOR xcnt := 0 TO SIZEOF(statusButtonActiv) - 1 DO
			statusButtonActiv[xcnt] := 1;
 			statusButtonInactiv[xcnt] := 0;
		END_FOR
		statusButtonActiv[6] := 0;
 		statusButtonInactiv[6] := 1;
	ELSIF (safeRemoteControl_0.SafeLOGICStatus.NumberOfUDIDMismatches > 4 AND safeRemoteControl_0.SafeLOGICStatus.Scanning = 0) THEN
		FOR xcnt := 0 TO SIZEOF(statusButtonActiv) - 1 DO
			statusButtonActiv[xcnt] := 1;
 			statusButtonInactiv[xcnt] := 0;
		END_FOR
		statusButtonActiv[7] := 0;
 		statusButtonInactiv[7] := 1;
	ELSIF (safeRemoteControl_0.SafeLOGICStatus.NumberOfDifferentFirmware <> 0 AND safeRemoteControl_0.SafeLOGICStatus.Scanning = 0) THEN
		FOR xcnt := 0 TO SIZEOF(statusButtonActiv) - 1 DO
			statusButtonActiv[xcnt] := 1;
 			statusButtonInactiv[xcnt] := 0;
		END_FOR
		statusButtonActiv[11] := 0;
 		statusButtonInactiv[11] := 1;
	ELSE
		FOR xcnt := 0 TO SIZEOF(statusButtonActiv) - 1 DO
			statusButtonActiv[xcnt] := 1;
 			statusButtonInactiv[xcnt] := 0;
		END_FOR
	END_IF
	(* status text - MXCHG *)
	IF (safeRemoteControl_0.SafeLOGICStatus.LedTestActive = 1) THEN
		indexMxchgLed := 40;
	ELSIF (safeRemoteControl_0.SafeLOGICStatus.Scanning = 1) THEN
		indexMxchgLed := 30;
	ELSIF (safeRemoteControl_0.SafeLOGICStatus.NumberOfUDIDMismatches = 1) THEN
		indexMxchgLed := 1;
	ELSIF (safeRemoteControl_0.SafeLOGICStatus.NumberOfUDIDMismatches = 2) THEN
		indexMxchgLed := 2;
	ELSIF (safeRemoteControl_0.SafeLOGICStatus.NumberOfUDIDMismatches = 3) THEN
		indexMxchgLed := 3;
	ELSIF (safeRemoteControl_0.SafeLOGICStatus.NumberOfUDIDMismatches = 4) THEN
		indexMxchgLed := 4;
	ELSIF (safeRemoteControl_0.SafeLOGICStatus.NumberOfUDIDMismatches > 4) THEN
		indexMxchgLed := 5;
	ELSIF (safeRemoteControl_0.SafeLOGICStatus.NumberOfMissingModules <> 0) THEN
		indexMxchgLed := 20;
	ELSIF (safeRemoteControl_0.SafeLOGICStatus.NumberOfUDIDMismatches = 0) THEN
		indexMxchgLed := 10;
	END_IF
	(* status text - FW-ACKN *)
	IF (safeRemoteControl_0.SafeLOGICStatus.SafeKEYChanged = 0 AND safeRemoteControl_0.SafeLOGICStatus.NumberOfDifferentFirmware = 0) THEN
		indexFwAcknLed := 10;
	ELSIF (safeRemoteControl_0.SafeLOGICStatus.SafeKEYChanged = 1) THEN
		indexFwAcknLed := 1;
	ELSIF (safeRemoteControl_0.SafeLOGICStatus.NumberOfDifferentFirmware <> 0) THEN
		indexFwAcknLed := 2;
	END_IF
	(* status text - FAIL *)
	IF (safeRemoteControl_0.SafeLOGICStatus.FailSafe <> 16#55) THEN
		indexFAILLed := 2;
	ELSIF (safeRemoteControl_0.SafeLOGICStatus.openSAFETYstate = 0) THEN
		indexFAILLed := 0;
	ELSIF (safeRemoteControl_0.SafeLOGICStatus.openSAFETYstate = 1) THEN
		indexFAILLed := 1;
	END_IF
	(* status text - R/E *)
	indexRELed := safeRemoteControl_0.SafeLOGICStatus.SafeOSState;

	(****************************************************************************************************************************************)
	(****************************************************************************************************************************************)
	(****************************************************************************************************************************************)
	(* show dialog to ackn command *)
	IF (dialogApplication = 1) THEN
		statusDialog := 0;
		dialogApplication := 0;
		indexButtonLeft := 0;
		indexButtonRight := 1;
		indexHeaderText := 1;
		indexMessageText := 10;
	END_IF

	(* if dialog is ackn unlock application *)
	IF (dialogButtonLeft = 1 AND indexHeaderText = 1) THEN
		appcmd1.Unlock := 1;
		dialogButtonLeft := 0;
		statusDialog := 1;
	ELSIF (dialogButtonRight = 1 AND indexHeaderText = 1) THEN
		appcmd1.Unlock := 2;
		dialogButtonRight := 0;
		statusDialog := 1;
	END_IF

	(* convert application CRC to HEX string *)
	itoahex(safeDownloadApplication_0.ApplicationCRC, ADR(visuApplicationCRC));

	safeDownloadApplication_0(SafeLOGICID := appcmd1.ApplicationID, Execute := executeapp1, pCommandData := ADR(appcmd1));

	(* show unlock button *)
	IF (safeDownloadApplication_0.UnlockRequired = 1) THEN
		statusButtonUnlockApp := 0;
	ELSE
		appcmd1.Unlock := 0;
		statusButtonUnlockApp := 1;
	END_IF

	(****************************************************************************************************************************************)
	(****************************************************************************************************************************************)
	(****************************************************************************************************************************************)
	(* disable machine options *)
	IF (visuEnableMachineOptions = FALSE) THEN
		datacmd1.pMachineOptionsInput := 0;
	ELSE
		datacmd1.pMachineOptionsInput := ADR(dataMachineOptionsBitInput);
	END_IF

	(* disable module flags *)
	IF (visuEnableModuleFlags = FALSE) THEN
		datacmd1.pModuleFlagsInput := 0;
	ELSE
		datacmd1.pModuleFlagsInput := ADR(dataModuleFlagsInput);
	END_IF

	(* Machine Option Bit #000 *)
	IF (visuMachineOptionsBitInput[0] = 1) THEN
		dataMachineOptionsBitInput.BitData[0].0 := 1;
	ELSE
		dataMachineOptionsBitInput.BitData[0].0 := 0;
	END_IF
	(* Machine Option Bit #001 *)
	IF (visuMachineOptionsBitInput[1] = 1) THEN
		dataMachineOptionsBitInput.BitData[0].1 := 1;
	ELSE
		dataMachineOptionsBitInput.BitData[0].1 := 0;
	END_IF
	(* Machine Option Bit #002 *)
	IF (visuMachineOptionsBitInput[2] = 1) THEN
		dataMachineOptionsBitInput.BitData[0].2 := 1;
	ELSE
		dataMachineOptionsBitInput.BitData[0].2 := 0;
	END_IF
	(* Optional Flag Module #1 *)
	IF (visuModuleFlagsOptionalInput[1] = 1) THEN
		dataModuleFlagsInput.Optional[0].1 := 1;
	ELSE
		dataModuleFlagsInput.Optional[0].1 := 0;
	END_IF
	(* Optional Flag Module #2 *)
	IF (visuModuleFlagsOptionalInput[2] = 1) THEN
		dataModuleFlagsInput.Optional[0].2 := 1;
	ELSE
		dataModuleFlagsInput.Optional[0].2 := 0;
	END_IF
	(* Startup Flag Module #1 *)
	IF (visuModuleFlagsStartupInput[1] = 1) THEN
		dataModuleFlagsInput.Startup[0].1 := 1;
	ELSE
		dataModuleFlagsInput.Startup[0].1 := 0;
	END_IF
	(* Startup Flag Module #2 *)
	IF (visuModuleFlagsStartupInput[2] = 1) THEN
		dataModuleFlagsInput.Startup[0].2 := 1;
	ELSE
		dataModuleFlagsInput.Startup[0].2 := 0;
	END_IF
	(* Not_Present Flag Module #1 *)
	IF (visuModuleFlagsNotPresentInput[1] = 1) THEN
		dataModuleFlagsInput.NotPresent[0].1 := 1;
	ELSE
		dataModuleFlagsInput.NotPresent[0].1 := 0;
	END_IF
	(* Not_Present Flag Module #2 *)
	IF (visuModuleFlagsNotPresentInput[2] = 1) THEN
		dataModuleFlagsInput.NotPresent[0].2 := 1;
	ELSE
		dataModuleFlagsInput.NotPresent[0].2 := 0;
	END_IF

	(* Ackn Machine Option Bit #000 *)
	IF (visuAcknMachineOptions[0] = 1) THEN
		dataAcknMachineOptions.AcknBitOptions[0].0 := 1;
	ELSE
		dataAcknMachineOptions.AcknBitOptions[0].0 := 0;
	END_IF
	(* Ackn Machine Option Bit #001 *)
	IF (visuAcknMachineOptions[1] = 1) THEN
		dataAcknMachineOptions.AcknBitOptions[0].1 := 1;
	ELSE
		dataAcknMachineOptions.AcknBitOptions[0].1 := 0;
	END_IF
	(* Ackn Machine Option Bit #002 *)
	IF (visuAcknMachineOptions[2] = 1) THEN
		dataAcknMachineOptions.AcknBitOptions[0].2 := 1;
	ELSE
		dataAcknMachineOptions.AcknBitOptions[0].2 := 0;
	END_IF

	(* show dialog to ackn command *)
	IF (dialogData = 1) THEN
		statusDialog := 0;
		dialogData := 0;
		indexButtonLeft := 0;
		indexButtonRight := 1;
		indexHeaderText := 2;
		indexMessageText := 11;
	END_IF

	(* if dialog is ackn unlock data *)
	IF (dialogButtonLeft = 1 AND indexHeaderText = 2) THEN
		datacmd1.Unlock := 1;
		dialogButtonLeft := 0;
		statusDialog := 1;
	ELSIF (dialogButtonRight = 1 AND indexHeaderText = 2) THEN
		datacmd1.Unlock := 2;
		dialogButtonRight := 0;
		statusDialog := 1;
	END_IF

	safeDownloadData_0(SafeLOGICID := visuUsedSLIDData, Execute := executedata1, Type:= safeDATA_TYPE_MAOP, pCommandData := ADR(datacmd1));

	(* data compare failed *)
	IF (safeDownloadData_0.StatusID = safeERR_DL_COMPARE_FAILED) THEN
		indexCompareTextData := 2;
	ELSE
		indexCompareTextData := 0;
	END_IF

	IF (safeDownloadData_0.UnlockRequired = 1) THEN
		(* data compare successful *)
		indexCompareTextData := 1;
		IF (datacmd1.pDeviceListOutput <> 0 AND datacmd1.NumberDevicesOutput <> 0) THEN
			pDeviceListOut ACCESS datacmd1.pDeviceListOutput;

			(* device #1 *)
			visuDeviceListOutput[0].SADR := pDeviceListOut[0].SADR;
			brsmemcpy(ADR(visuDeviceListOutput[0].UDID_High), ADR(pDeviceListOut[0].UDID[0]), 2);
			(* swap UDID *)
			visuDeviceListOutput[0].UDID_High := swapUINT(visuDeviceListOutput[0].UDID_High);
			brsmemcpy(ADR(visuDeviceListOutput[0].UDID_Low), ADR(pDeviceListOut[0].UDID[2]), 4);
			(* swap UDID *)
			visuDeviceListOutput[0].UDID_Low := swapUDINT(visuDeviceListOutput[0].UDID_Low);
			(* device #2 *)
			visuDeviceListOutput[1].SADR := pDeviceListOut[1].SADR;
			brsmemcpy(ADR(visuDeviceListOutput[1].UDID_High), ADR(pDeviceListOut[1].UDID[0]), 2);
			(* swap UDID *)
			visuDeviceListOutput[1].UDID_High := swapUINT(visuDeviceListOutput[1].UDID_High);
			brsmemcpy(ADR(visuDeviceListOutput[1].UDID_Low), ADR(pDeviceListOut[1].UDID[2]), 4);
			(* swap UDID *)
			visuDeviceListOutput[1].UDID_Low := swapUDINT(visuDeviceListOutput[1].UDID_Low);
		END_IF

		IF (datacmd1.pMachineOptionsOutput <> 0) THEN
			pMachineOptionsBitOut ACCESS datacmd1.pMachineOptionsOutput;

			(* Machine Option Bit #000 *)
			IF (pMachineOptionsBitOut.BitData[0].0 = 1) THEN
				visuMachineOptionsBitOutput[0] := 1;
			END_IF
			(* Machine Option Bit #001 *)
			IF (pMachineOptionsBitOut.BitData[0].1 = 1) THEN
				visuMachineOptionsBitOutput[1] := 1;
			END_IF
			(* Machine Option Bit #002 *)
			IF (pMachineOptionsBitOut.BitData[0].2 = 1) THEN
				visuMachineOptionsBitOutput[2] := 1;
			END_IF
		END_IF

		IF (datacmd1.pModuleFlagsOutput <> 0) THEN
			pModuleFlagsOut ACCESS datacmd1.pModuleFlagsOutput;

			(* Optional Flag Module #1 *)
			IF (pModuleFlagsOut.Optional[0].1 = 1) THEN
				visuModuleFlagsOptionalOutput[1] := 1;
			END_IF
			(* Optional Flag Module #2 *)
			IF (pModuleFlagsOut.Optional[0].2 = 1) THEN
				visuModuleFlagsOptionalOutput[2] := 1;
			END_IF
			(* Startup Flag Module #1 *)
			IF (pModuleFlagsOut.Startup[0].1 = 1) THEN
				visuModuleFlagsStartupOutput[1] := 1;
			END_IF
			(* Startup Flag Module #2 *)
			IF (pModuleFlagsOut.Startup[0].2 = 1) THEN
				visuModuleFlagsStartupOutput[2] := 1;
			END_IF
			(* Not_Present Flag Module #1 *)
			IF (pModuleFlagsOut.NotPresent[0].1 = 1) THEN
				visuModuleFlagsNotPresentOutput[1] := 1;
			END_IF
			(* Not_Present Flag Module #2 *)
			IF (pModuleFlagsOut.NotPresent[0].2 = 1) THEN
				visuModuleFlagsNotPresentOutput[2] := 1;
			END_IF
		END_IF
		(* show ackn box *)
		statusAcknInfoData := 0;
		(* show unlock button unlocked if one ACK is set *)
		IF (visuAcknMachineOptions[0] = 1 OR visuAcknMachineOptions[1] = 1 OR visuAcknMachineOptions[2] = 1) THEN
			statusButtonUnlockData := 0;
		END_IF
	ELSIF (safeDownloadData_0.Done = 1 OR safeDownloadData_0.Error = 1) THEN
		(* reset visualization elements *)
		brsmemset(ADR(visuDeviceListOutput), 0, SIZEOF(visuDeviceListOutput));
		brsmemset(ADR(visuMachineOptionsBitOutput), 0, SIZEOF(visuMachineOptionsBitOutput));
		brsmemset(ADR(visuModuleFlagsOptionalOutput), 0, SIZEOF(visuModuleFlagsOptionalOutput));
		brsmemset(ADR(visuModuleFlagsStartupOutput), 0, SIZEOF(visuModuleFlagsStartupOutput));
		brsmemset(ADR(visuModuleFlagsNotPresentOutput), 0, SIZEOF(visuModuleFlagsNotPresentOutput));
		(* hide ackn box *)
		statusAcknInfoData := 1;
		(* hide unlock button *)
		datacmd1.Unlock := 0;
		statusButtonUnlockData := 1;
		(* reset ackn flags *)
		visuAcknMachineOptions[0] := 0;
		visuAcknMachineOptions[1] := 0;
		visuAcknMachineOptions[2] := 0;
	ELSE
		(* hide ackn box *)
		statusAcknInfoData := 1;
		(* hide unlock button *)
		datacmd1.Unlock := 0;
		statusButtonUnlockData := 1;
	END_IF

	(****************************************************************************************************************************************)
	(****************************************************************************************************************************************)
	(****************************************************************************************************************************************)
	(* Enable for INT set *)
	IF (visuEnableINTOptions <> 0) THEN
		datacmd2.pIntDataInput := ADR(visuIntInput);
		datacmd2.NumberIntInput := 1;
	ELSE
		datacmd2.pIntDataInput := 0;
		datacmd2.NumberIntInput := 0;
	END_IF
	(* Enable for UINT set *)
	IF (visuEnableUINTOptions <> 0) THEN
		datacmd2.pUintDataInput := ADR(visuUintInput);
		datacmd2.NumberUintInput := 1;
	ELSE
		datacmd2.pUintDataInput := 0;
		datacmd2.NumberUintInput := 0;
	END_IF
	(* Enable for DINT set *)
	IF (visuEnableDINTOptions <> 0) THEN
		datacmd2.pDintDataInput := ADR(visuDintInput);
		datacmd2.NumberDintInput := 1;
	ELSE
		datacmd2.pDintDataInput := 0;
		datacmd2.NumberDintInput := 0;
	END_IF
	(* Enable for UDINT set *)
	IF (visuEnableUDINTOptions <> 0) THEN
		datacmd2.pUdintDataInput := ADR(visuUdintInput);
		datacmd2.NumberUdintInput := 1;
	ELSE
		datacmd2.pUdintDataInput := 0;
		datacmd2.NumberUdintInput := 0;
	END_IF

	(* show dialog to ackn command *)
	IF (dialogExtData = 1) THEN
		statusDialog := 0;
		dialogExtData := 0;
		indexButtonLeft := 0;
		indexButtonRight := 1;
		indexHeaderText := 3;
		indexMessageText := 11;
	END_IF

	(* if dialog is ackn unlock data *)
	IF (dialogButtonLeft = 1 AND indexHeaderText = 3) THEN
		datacmd2.Unlock := 1;
		dialogButtonLeft := 0;
		statusDialog := 1;
	ELSIF (dialogButtonRight = 1 AND indexHeaderText = 3) THEN
		datacmd2.Unlock := 2;
		dialogButtonRight := 0;
		statusDialog := 1;
	END_IF

	safeDownloadData_1(SafeLOGICID := visuUsedSLIDData, Execute := executedata2, Type:= safeDATA_TYPE_EXTMAOP, pCommandData := ADR(datacmd2));

	(* data compare failed *)
	IF (safeDownloadData_1.StatusID = safeERR_DL_COMPARE_FAILED) THEN
		indexCompareTextExtData := 2;
	ELSE
		indexCompareTextExtData := 0;
	END_IF

	IF (safeDownloadData_1.UnlockRequired = 1) THEN
		(* data compare successful *)
		indexCompareTextExtData := 1;

		(* INT channels *)
		IF (datacmd2.pIntDataOutput <> 0 AND datacmd2.NumberIntOutput <> 0) THEN
			brsmemcpy(ADR(visuIntOutput), datacmd2.pIntDataOutput, SIZEOF(visuIntOutput));
		END_IF
		(* UINT channels *)
		IF (datacmd2.pUintDataOutput <> 0 AND datacmd2.NumberUintOutput <> 0) THEN
			brsmemcpy(ADR(visuUintOutput), datacmd2.pUintDataOutput, SIZEOF(visuUintOutput));
		END_IF
		(* DINT channels *)
		IF (datacmd2.pDintDataOutput <> 0 AND datacmd2.NumberDintOutput <> 0) THEN
			brsmemcpy(ADR(visuDintOutput), datacmd2.pDintDataOutput, SIZEOF(visuDintOutput));
		END_IF
		(* UDINT channels *)
		IF (datacmd2.pUdintDataOutput <> 0 AND datacmd2.NumberUdintOutput <> 0) THEN
			brsmemcpy(ADR(visuUdintOutput), datacmd2.pUdintDataOutput, SIZEOF(visuUdintOutput));
		END_IF
		(* show ackn box *)
		statusAcknInfoExtData := 0;
		(* show unlock button if one ACK is set *)
		IF (visuAcknExtData.AcknIntOptions[0] = 1 OR visuAcknExtData.AcknUintOptions[0] = 1 OR visuAcknExtData.AcknDintOptions[0] = 1 OR visuAcknExtData.AcknUdintOptions[0] = 1) THEN
			statusButtonUnlockExtData := 0;
		END_IF
	ELSIF (safeDownloadData_1.Done = 1 OR safeDownloadData_1.Error = 1) THEN
		(* reset visualization elements *)
		brsmemset(ADR(visuIntOutput), 0, SIZEOF(visuIntOutput));
		brsmemset(ADR(visuUintOutput), 0, SIZEOF(visuUintOutput));
		brsmemset(ADR(visuDintOutput), 0, SIZEOF(visuDintOutput));
		brsmemset(ADR(visuUdintOutput), 0, SIZEOF(visuUdintOutput));
		(* hide ackn box *)
		statusAcknInfoExtData := 1;
		(* hide unlock button *)
		datacmd2.Unlock := 0;
		statusButtonUnlockExtData := 1;
		(* reset ackn flags *)
		visuAcknExtData.AcknIntOptions[0] := 0;
		visuAcknExtData.AcknUintOptions[0] := 0;
		visuAcknExtData.AcknDintOptions[0] := 0;
		visuAcknExtData.AcknUdintOptions[0] := 0;
	ELSE
		(* hide ackn box *)
		statusAcknInfoExtData := 1;
		(* hide unlock button *)
		datacmd2.Unlock := 0;
		statusButtonUnlockExtData := 1;
	END_IF

	(****************************************************************************************************************************************)
	(****************************************************************************************************************************************)
	(****************************************************************************************************************************************)
	(* read UDID from SafeLOGIC-X *)
	IF slxused = 1 THEN
		readUDIDlowSLX(enable := 1, pDeviceName := ADR(Station), pChannelName := ADR('UDID_low'));

		IF readUDIDlowSLX.status = 0 THEN
			UDID_Low := readUDIDlowSLX.value;
		ELSIF readUDIDlowSLX.status <> 65535 THEN
			UDID_Low := 0;
		END_IF

		readUDIDhighSLX(enable := 1, pDeviceName := ADR(Station), pChannelName := ADR('UDID_high'));

		IF readUDIDhighSLX.status = 0 THEN
			UDID_High := UDINT_TO_UINT(readUDIDhighSLX.value);
		ELSIF readUDIDhighSLX.status <> 65535 THEN
			UDID_High := 0;
		END_IF

		(* hide / show visualization elements *)
		stautsSLXInformation := 0;
		statusSLInformation := 1;
	(* read UDID form SafeLOGIC *)
	ELSE
		readUDIDlowSL(enable := 1, pDevice := ADR(Interface), node := Node, index := 16#2000, subindex := 6, pData := ADR(UDID_Low), datalen := SIZEOF(UDID_Low));

		IF readUDIDlowSL.status <> 0 AND readUDIDlowSL.status <> 65535 THEN
			UDID_Low := 0;
		END_IF

		readUDIDhighSL(enable := 1, pDevice := ADR(Interface), node := Node, index := 16#2000, subindex := 7, pData := ADR(UDID_High), datalen := SIZEOF(UDID_High));

		IF readUDIDhighSL.status <> 0 AND readUDIDhighSL.status <> 65535 THEN
			UDID_High := 0;
		END_IF

		(* hide / show visualization elements *)
		stautsSLXInformation := 1;
		statusSLInformation := 0;
	END_IF

	(* convert UDID to HEX string *)
	itoahex(UDID_Low, ADR(visuUDID_Low));
	itoahex(UDID_High, ADR(visuUDID_High));

	(****************************************************************************************************************************************)
	(****************************************************************************************************************************************)
	(****************************************************************************************************************************************)
	(* write UDID for SafeLOGIC to command structure *)
	appcmd1.UDID_Low := UDID_Low;
	appcmd1.UDID_High := UDID_High;
	datacmd1.UDID_Low := UDID_Low;
	datacmd1.UDID_High := UDID_High;
	datacmd2.UDID_Low := UDID_Low;
	datacmd2.UDID_High := UDID_High;

END_PROGRAM
```

### gFeedi.ax
```
InitParameter (Version=5.08.2, NcSwId=ACP10)
  ACP10AXIS_typ:
    dig_in:
      level:
        reference = ncACTIV_HI
        pos_hw_end = ncACTIV_HI
        neg_hw_end = ncACTIV_HI
        trigger1 = ncACTIV_HI
        trigger2 = ncACTIV_HI
    encoder_if:
      parameter:
        count_dir = ncSTANDARD
        scaling:
          load:
            units = 12700
            rev_motor = 10
    limit:
      parameter:
        v_pos = 100000.0
        v_neg = 100000.0
        a1_pos = 500000.0
        a2_pos = 500000.0
        a1_neg = 500000.0
        a2_neg = 500000.0
        t_jolt = 0.0
        t_in_pos = 0.0
        pos_sw_end = 10000
        neg_sw_end = 0
        ds_warning = 200.0
        ds_stop = 200.0
        a_stop = 1.0E+30
        dv_stop = 0.0
        dv_stop_mode = ncOFF
    controller:
      mode = ncPOSITION
      position:
        kv = 400.0
        tn = 0.0
        t_predict = 0.0004
        t_total = 0.0004
        p_max = 1.0E+30
        i_max = 1.0E+30
      speed:
        kv = 0.6
        tn = 0.1
        t_filter = 0.0
        isq_filter1:
          type = ncOFF
          a0 = 0.0
          a1 = 0.0
          b0 = 0.0
          b1 = 0.0
          b2 = 0.0
          c0_par_id = 0
          c1_par_id = 0
        isq_filter2:
          type = ncOFF
          a0 = 0.0
          a1 = 0.0
          b0 = 0.0
          b1 = 0.0
          b2 = 0.0
          c0_par_id = 0
          c1_par_id = 0
        isq_filter3:
          type = ncOFF
          a0 = 0.0
          a1 = 0.0
          b0 = 0.0
          b1 = 0.0
          b2 = 0.0
          c0_par_id = 0
          c1_par_id = 0
      uf:
        type = ncLINEAR
        auto_config = ncOFF
        u0 = 0.0
        un = 0.0
        fn = 0.0
        k_f_slip = 0.0
      ff:
        mode = ncSTANDARD
        torque_load = 0.0
        torque_pos = 0.0
        torque_neg = 0.0
        kv_torque = 0.0
        inertia = 0.0
        t_filter_a = 0.0
      fb:
        mode = ncSTANDARD
        speed_mix_ratio = 0.0
        speed_kv = 2.0
      model:
        mass1:
          inertia = 0.0
          viscous_friction = 0.0
        mass2:
          inertia = 0.0
          viscous_friction = 0.0
          stiffness = 0.0
          damping = 0.0
    move:
      stop:
        parameter[0]:
          decel_ramp = ncA_LIMIT
          controller = ncON
        parameter[1]:
          decel_ramp = ncA_LIMIT
          controller = ncON
        parameter[2]:
          decel_ramp = ncA_LIMIT
          controller = ncON
        parameter[3]:
          decel_ramp = ncA_LIMIT
          controller = ncON
        quickstop:
          decel_ramp = ncA_LIMIT
          t_jolt = 0.0
        drive_error:
          decel_ramp = ncA_LIMIT
      homing:
        parameter:
          s = 0
          v_switch = 5000.0
          v_trigger = 500.0
          a = 50000.0
          mode = ncDIRECT
          edge_sw = ncPOSITIVE
          start_dir = ncPOSITIVE
          trigg_dir = ncPOSITIVE
          ref_pulse = ncOFF
          fix_dir = ncOFF
          tr_s_block = 0.0
          torque_lim = 0.0
          ds_block = 0.0
          ds_stop = 0.0
      basis:
        parameter:
          v_pos = 635.0
          v_neg = 635.0
          a1_pos = 36000.0
          a2_pos = 36000.0
          a1_neg = 36000.0
          a2_neg = 36000.0
    message:
      text:
        parameter:
          format = ncBREAK
          columns = 80
          data_modul = acp10etxen
```

### Program Logical/HMI/HMIControl (IEC)

#### Cyclic.ld
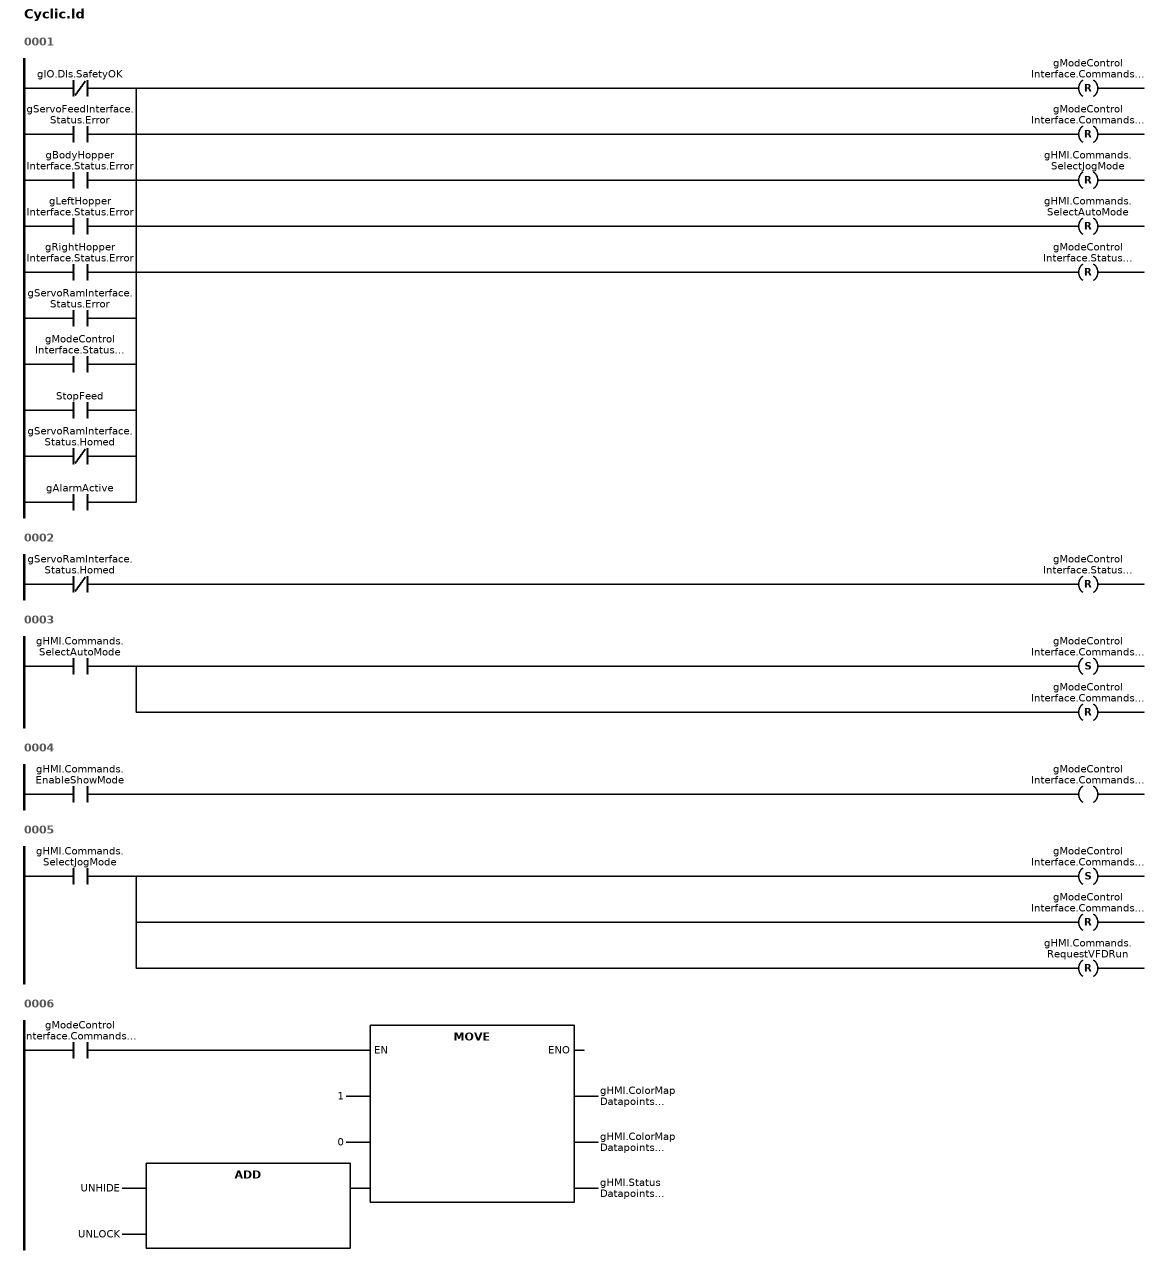
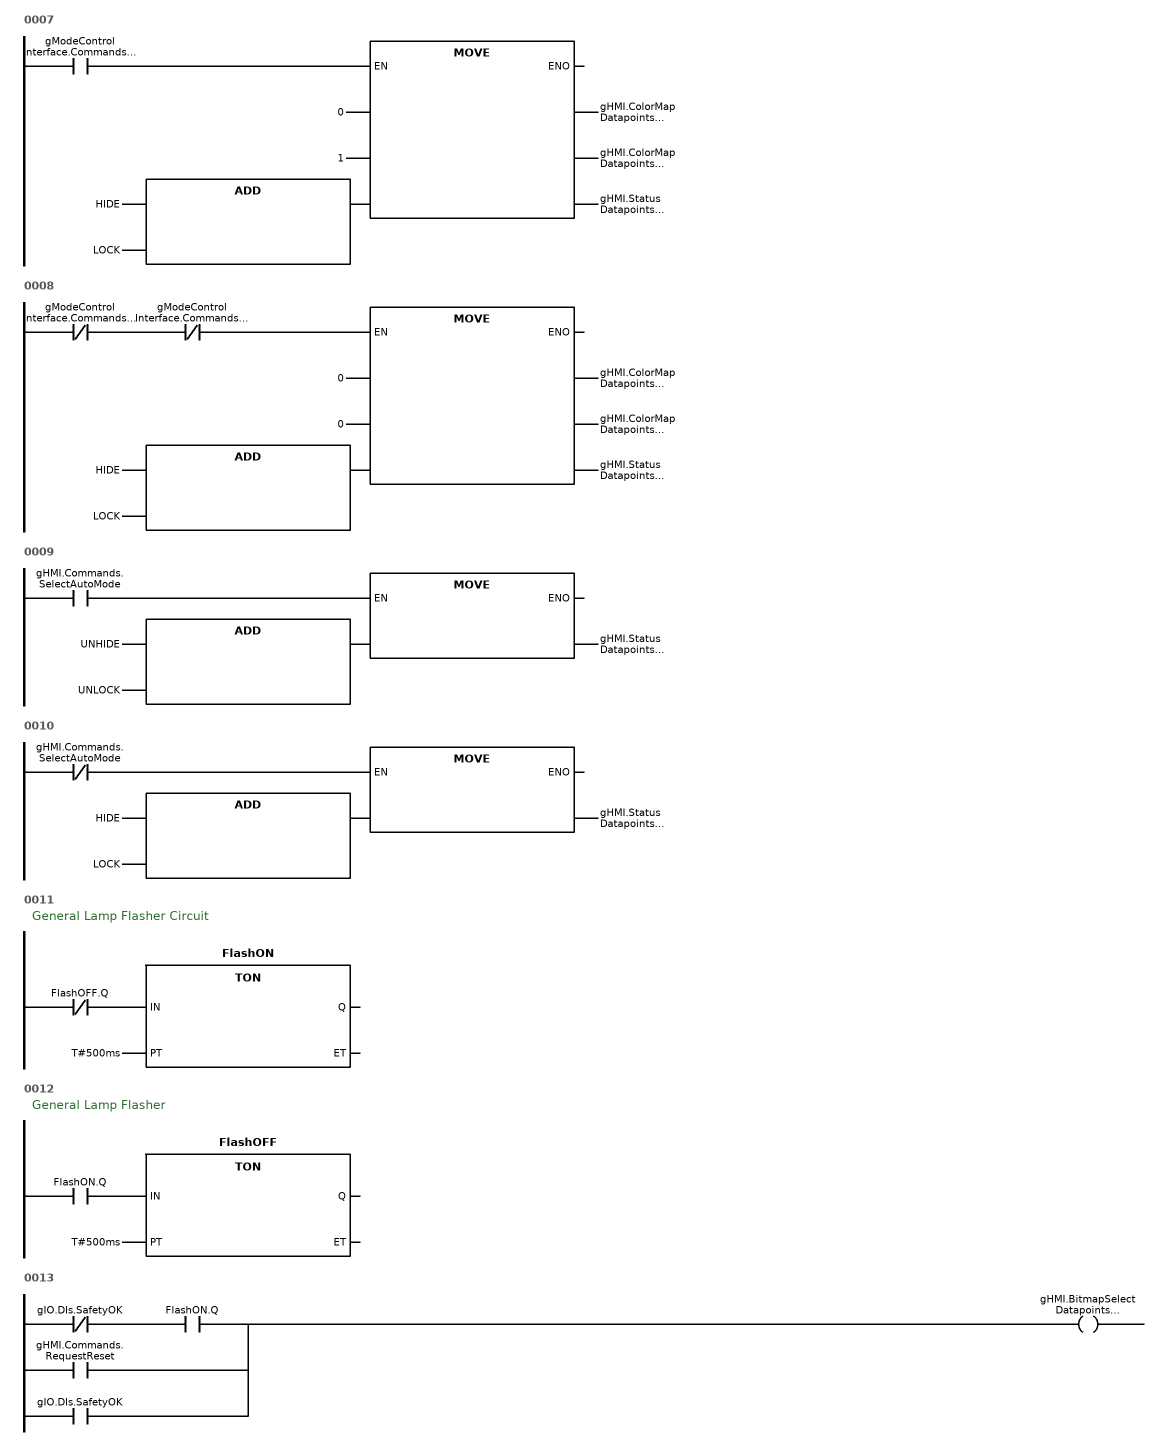
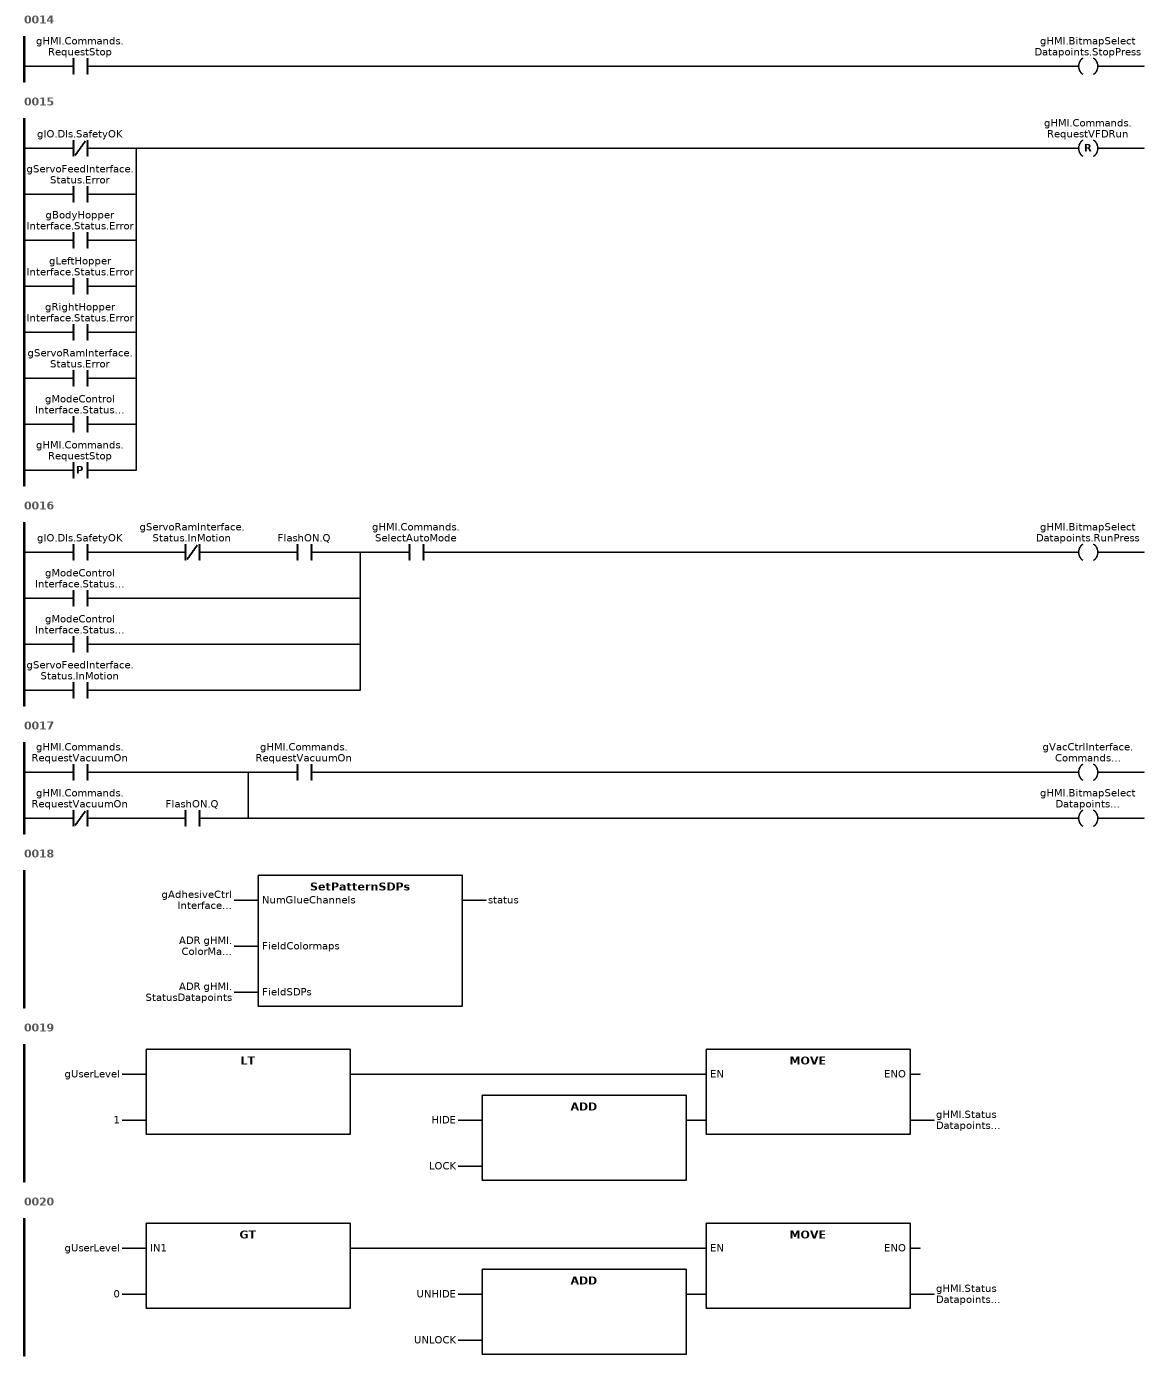
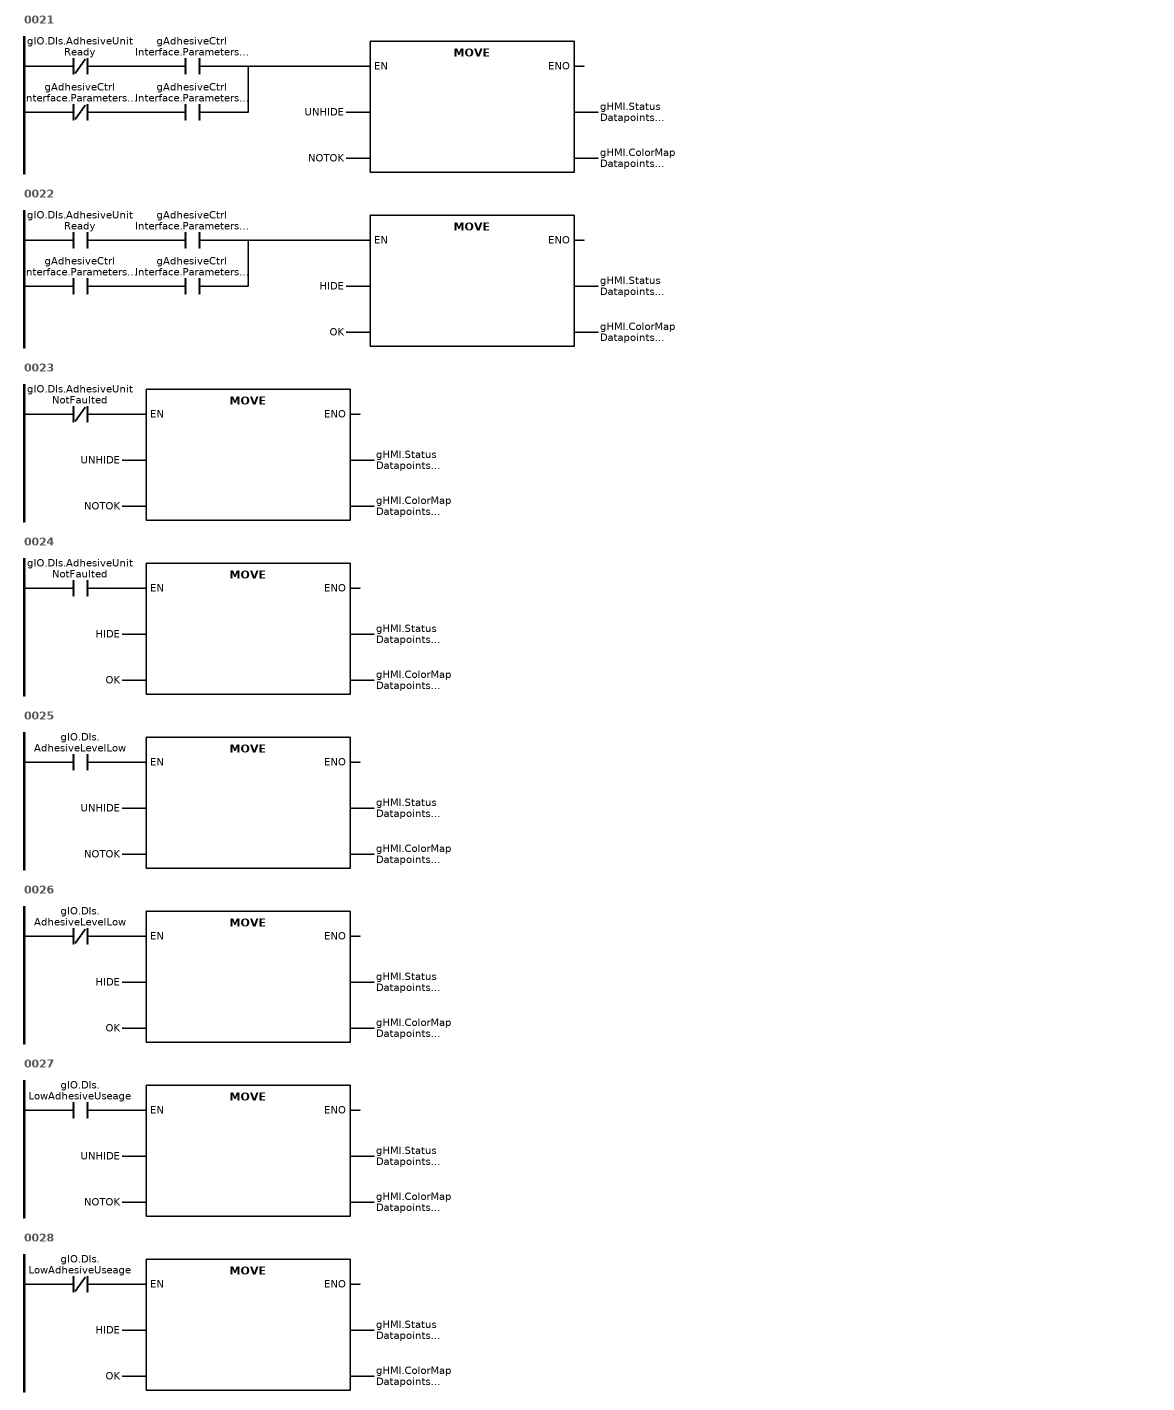
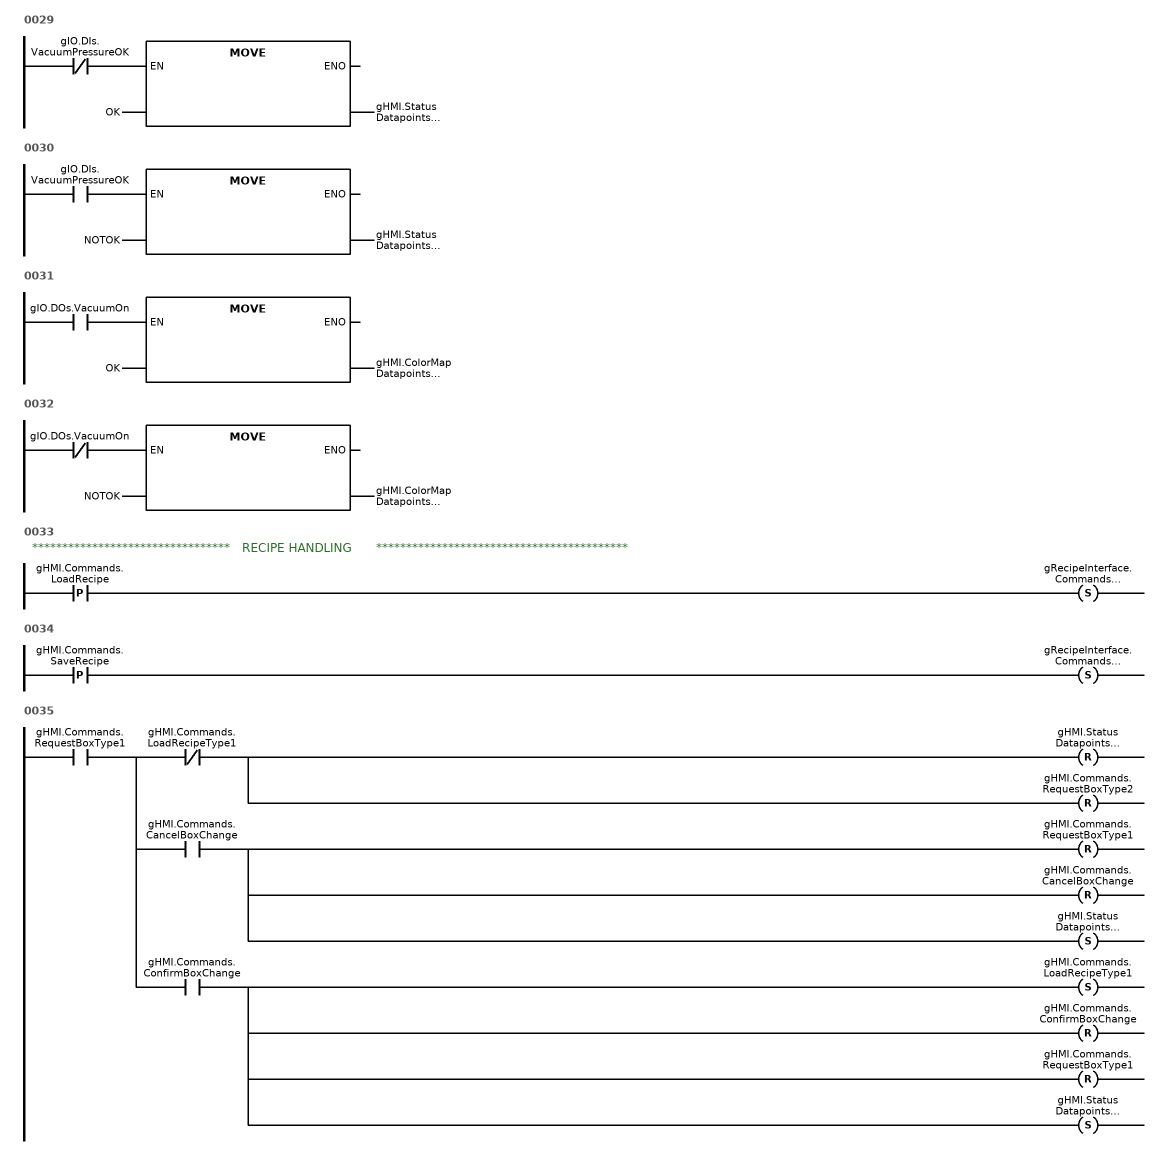
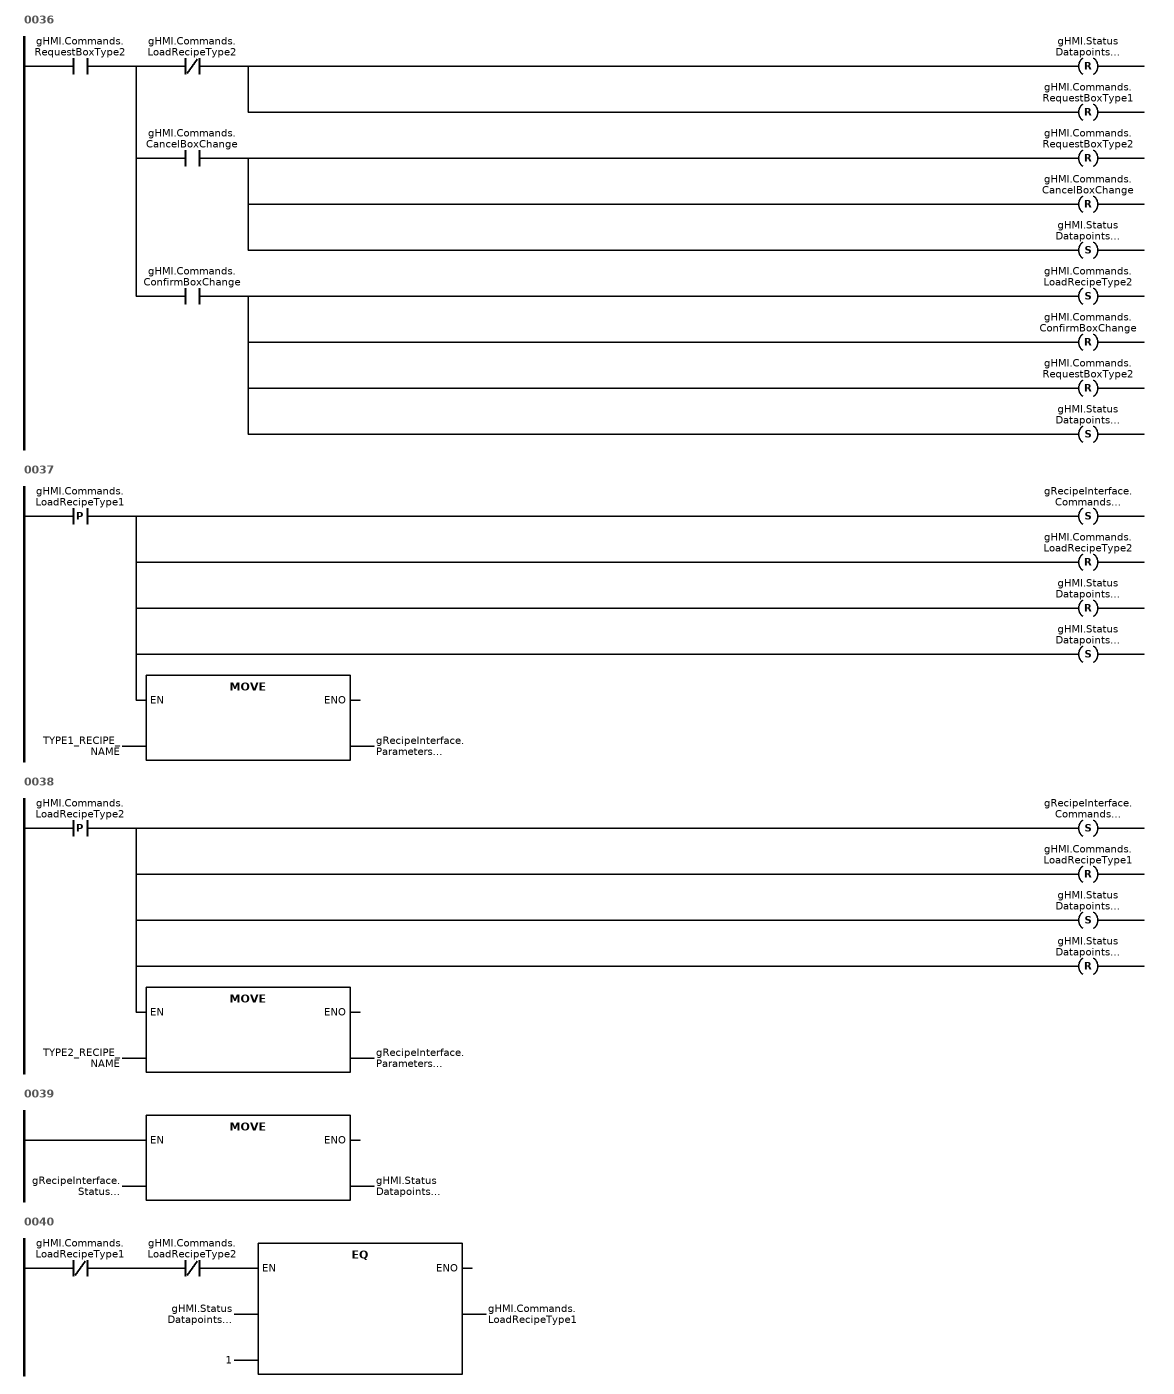
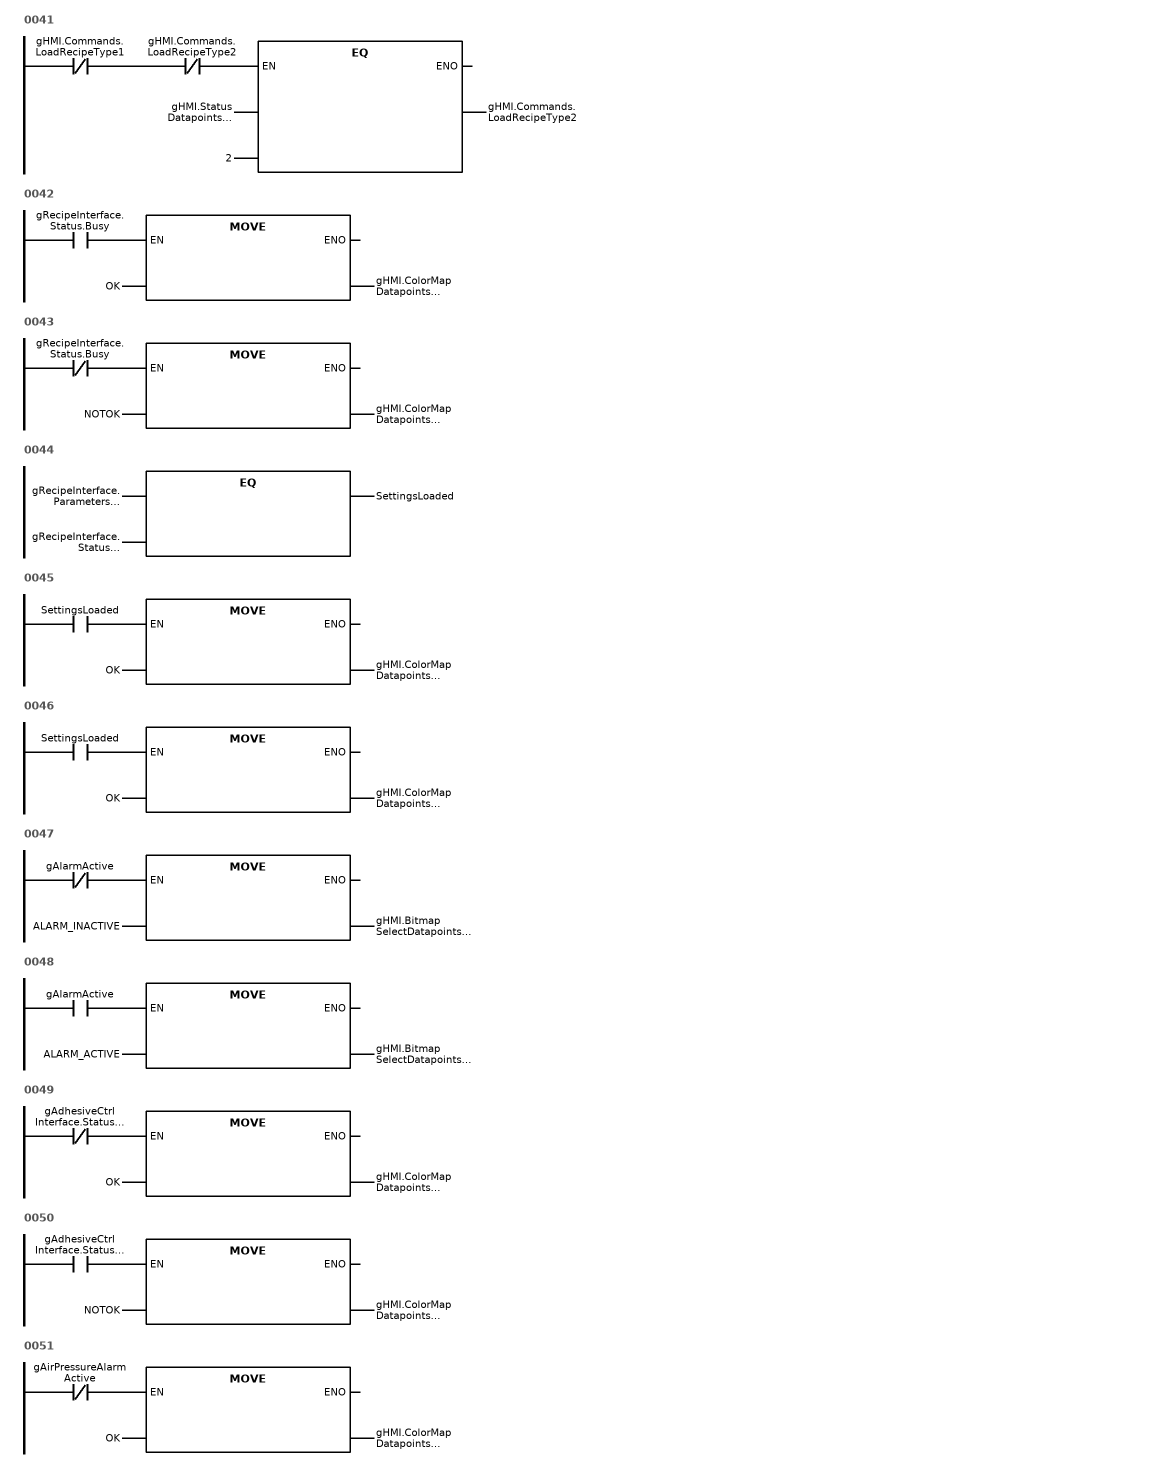
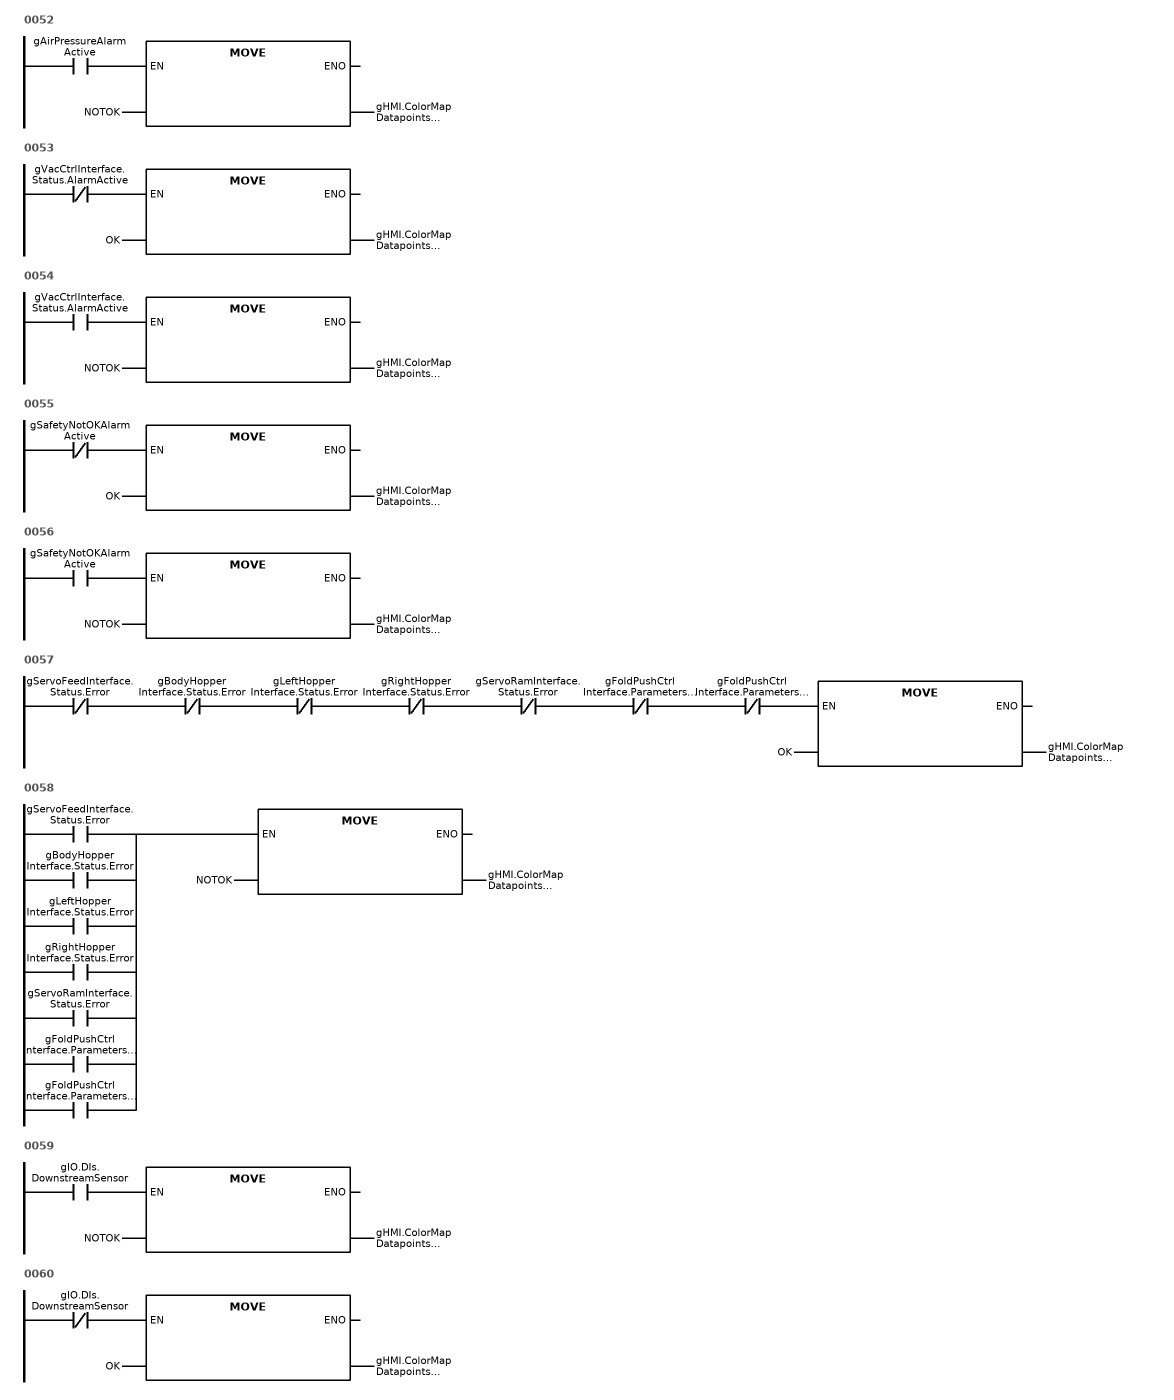
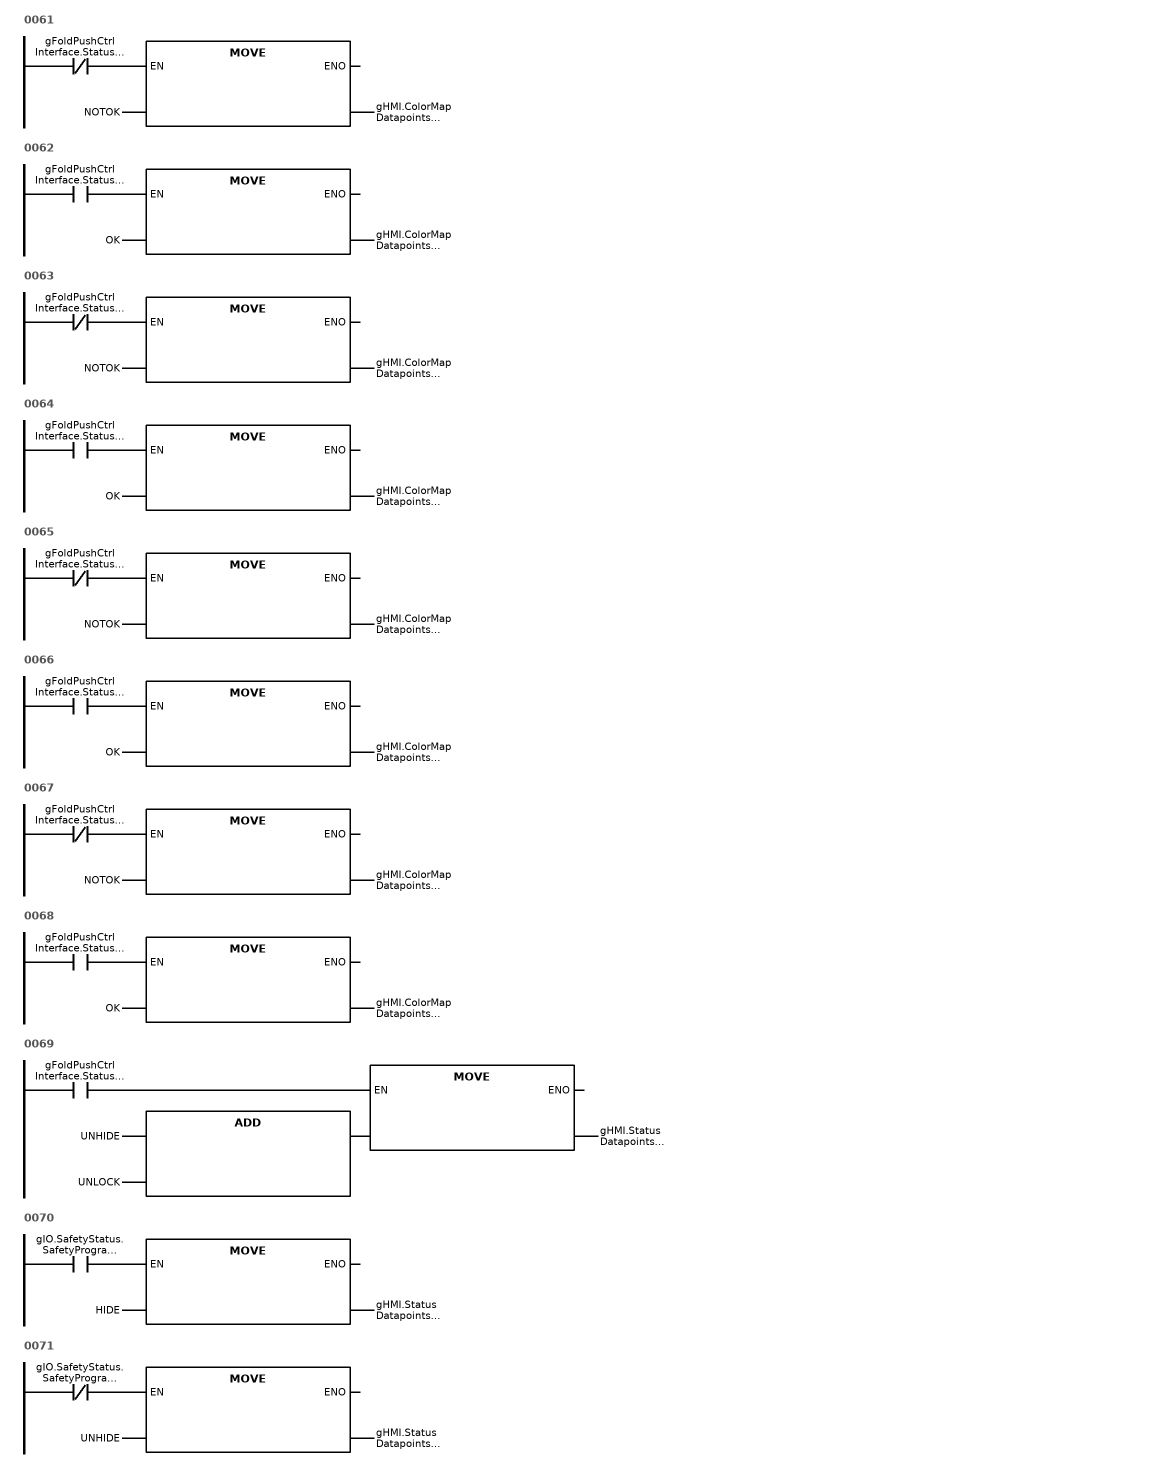
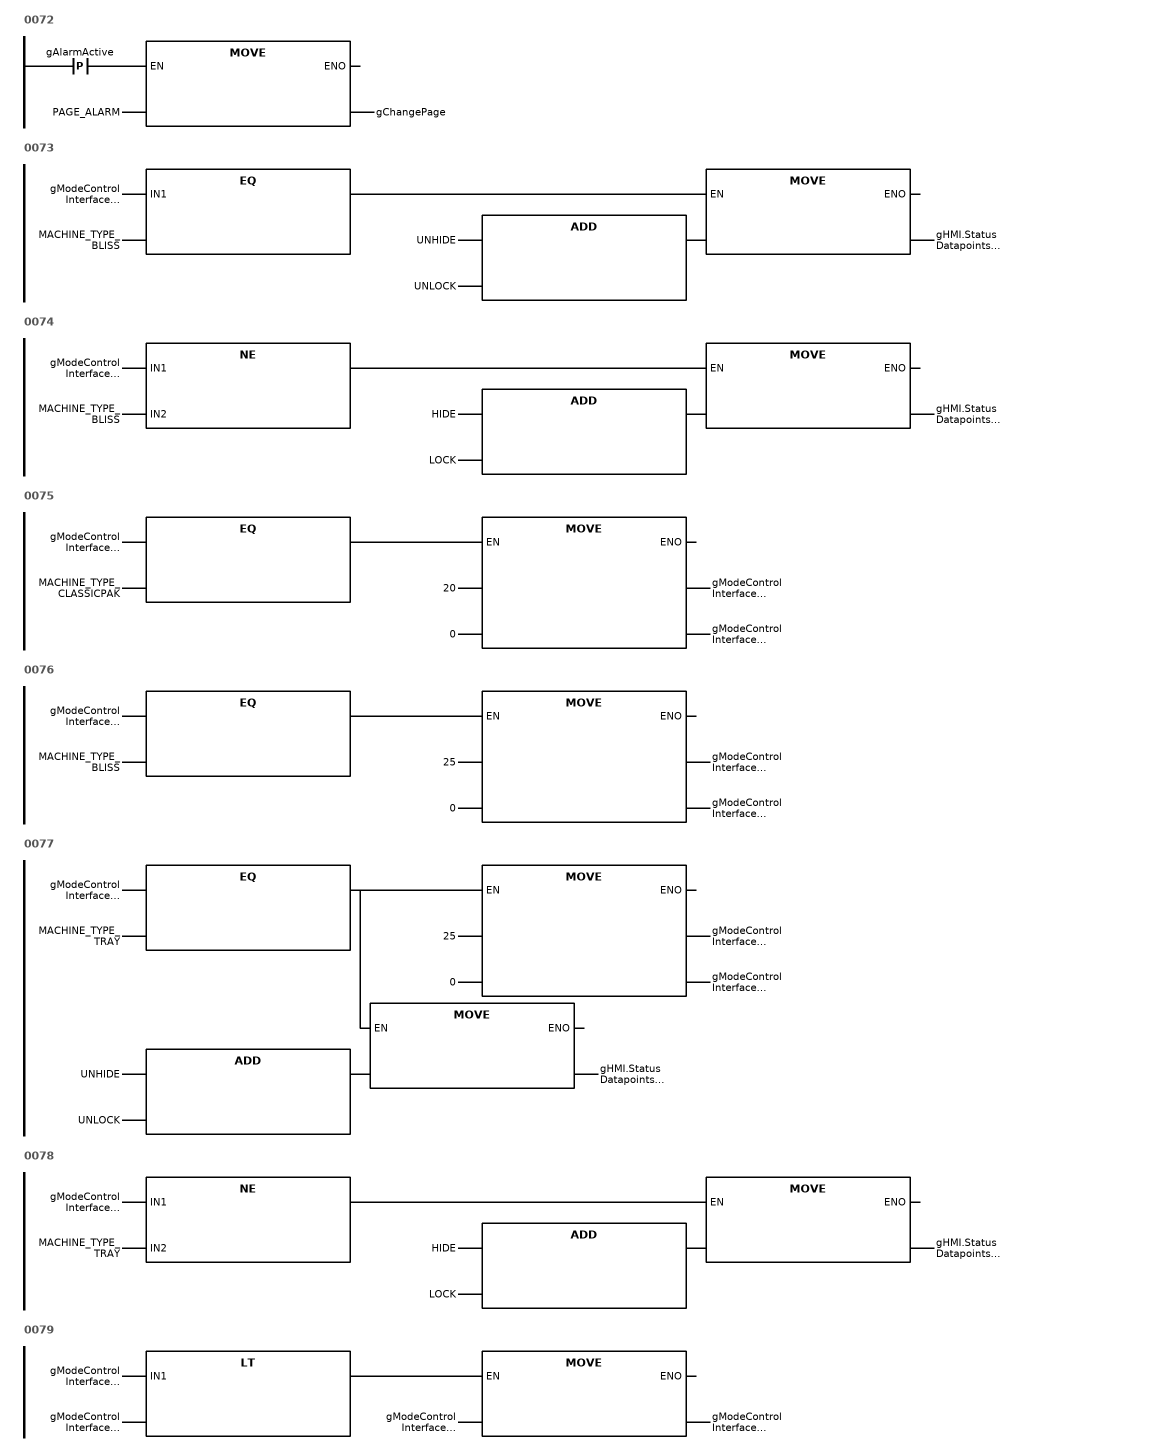
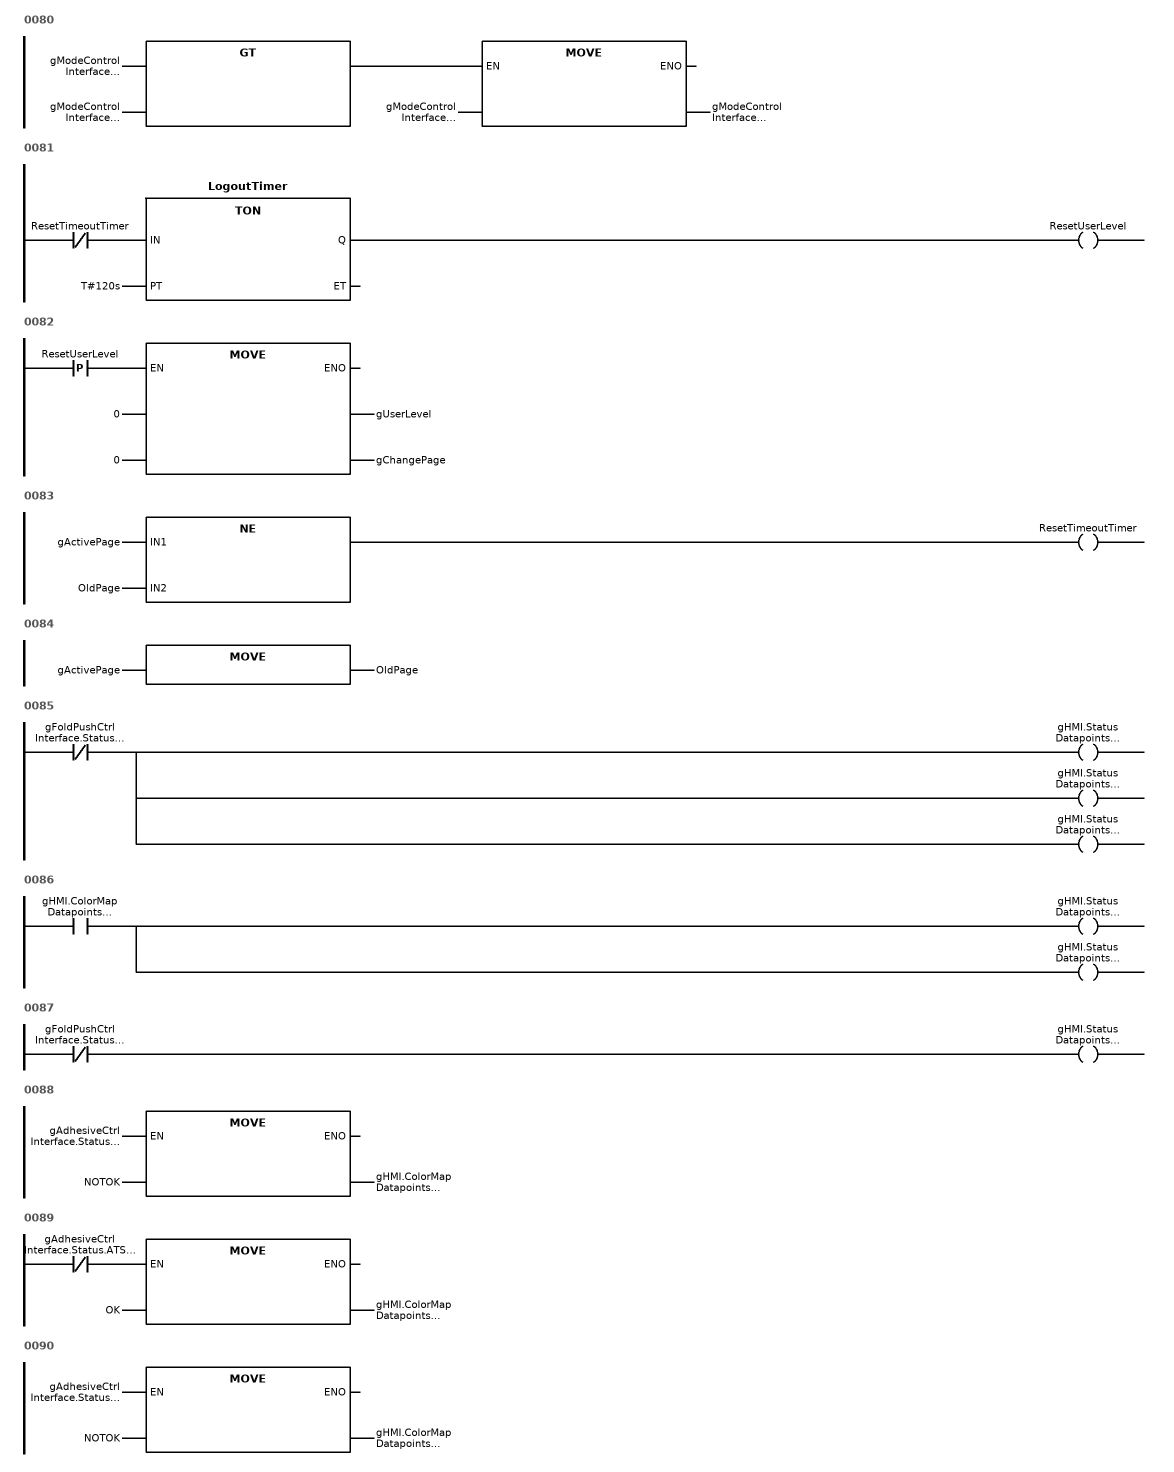
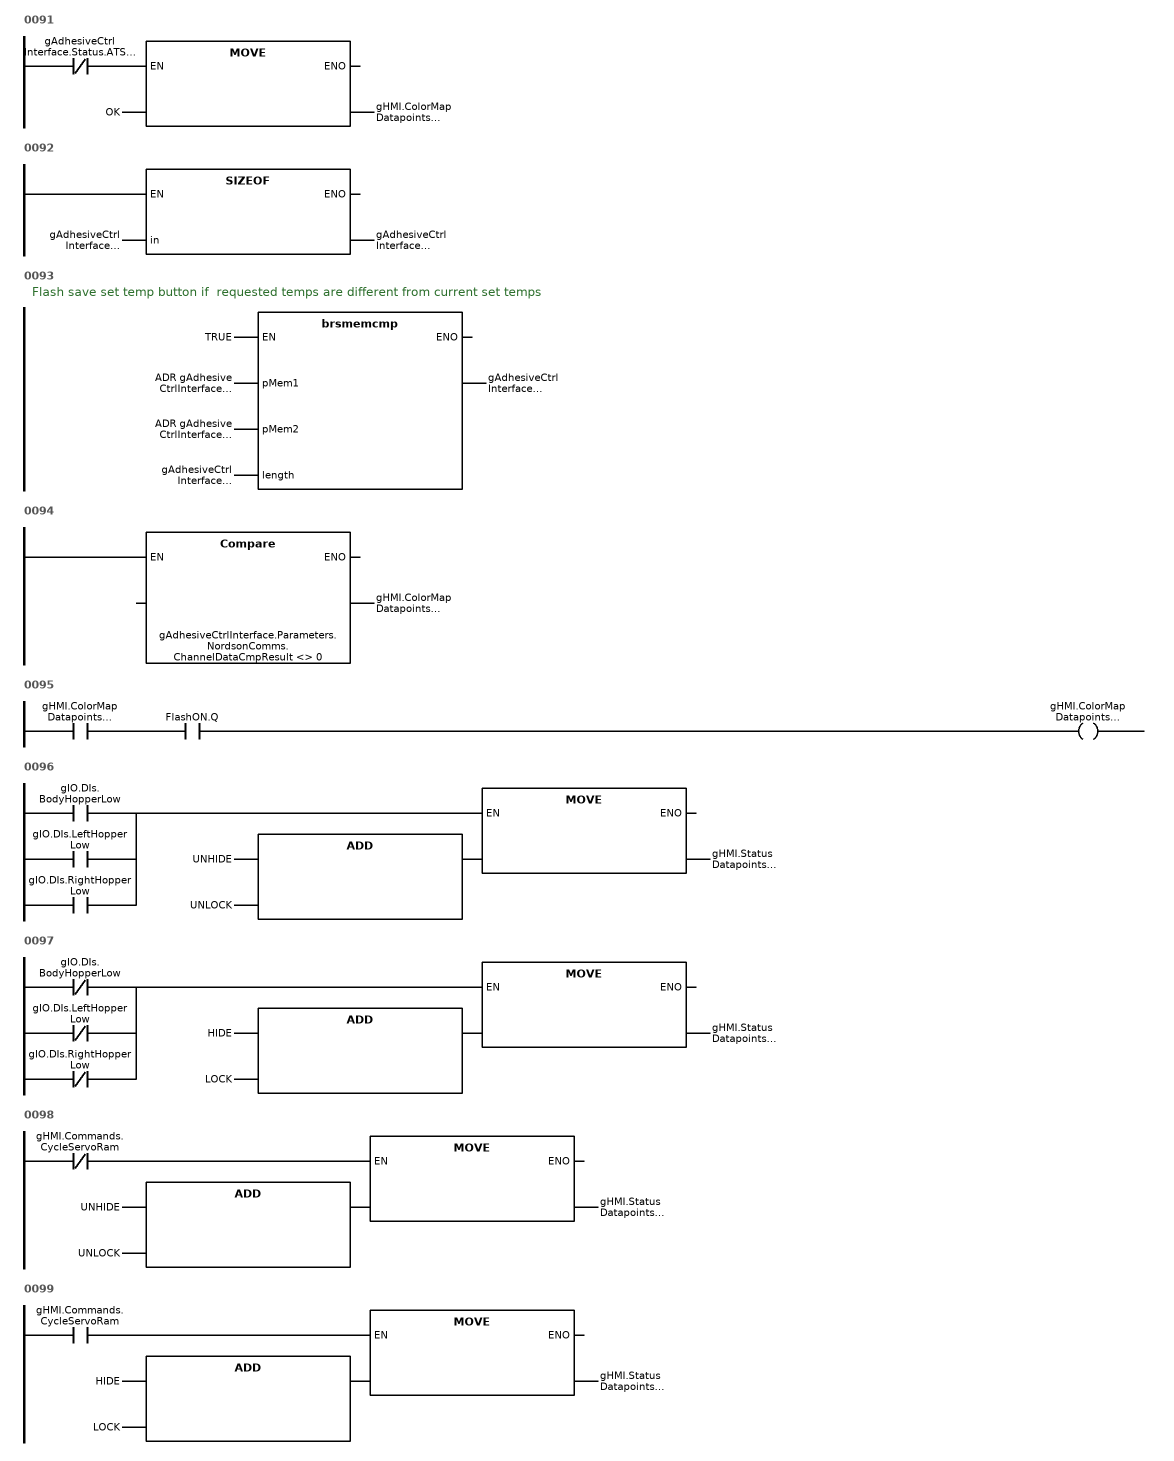
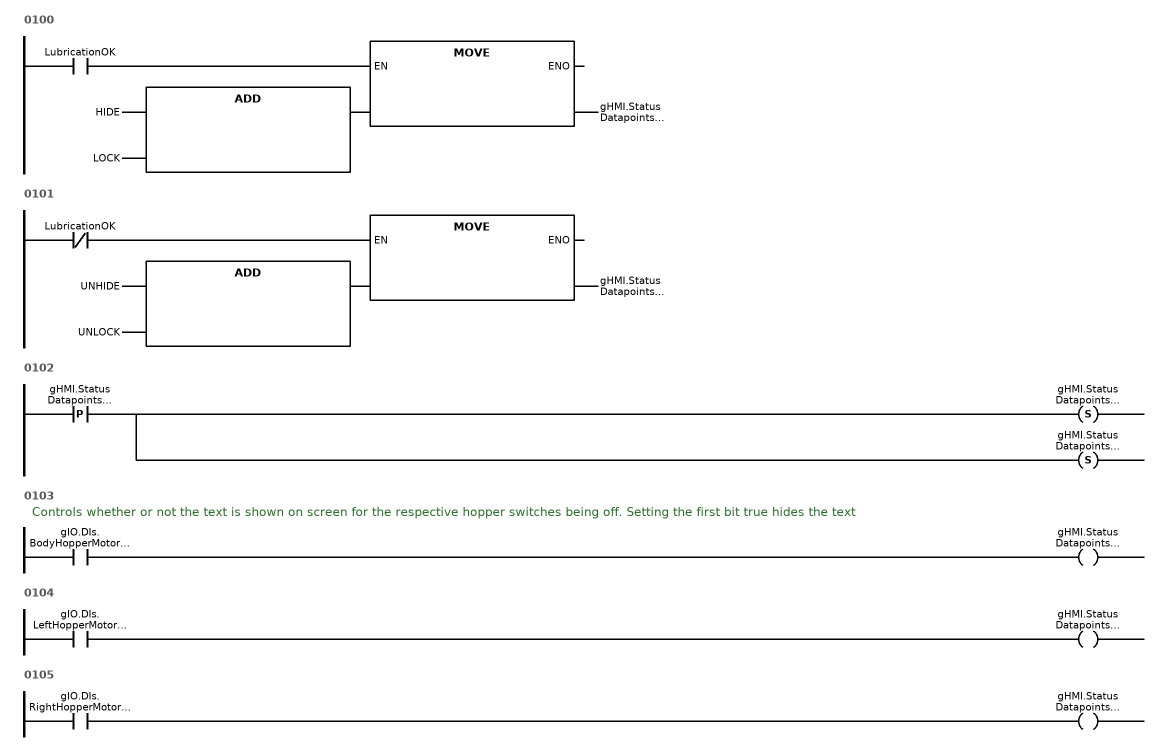
Ladder, written as Structured Text:
```iecst
PROGRAM _CYCLIC
VAR
    _p1 : BOOL;
    _p2 : BOOL;
    _p3 : BOOL;
    _p4 : BOOL;
    _e5 : R_TRIG;
    _p6 : BOOL;
    _p7 : BOOL;
    _p8 : BOOL;
    _p9 : BOOL;
    _e10 : R_TRIG;
    _e11 : R_TRIG;
    _p12 : BOOL;
    _p13 : BOOL;
    _p14 : BOOL;
    _p15 : BOOL;
    _p16 : BOOL;
    _p17 : BOOL;
    _p18 : BOOL;
    _p19 : BOOL;
    _e20 : R_TRIG;
    _e21 : R_TRIG;
    _p22 : BOOL;
    _p23 : BOOL;
    _e24 : R_TRIG;
    _t25 : BOOL;
    _t26 : BOOL;
    _t27 : BOOL;
    _p28 : BOOL;
    _p29 : BOOL;
    _e30 : R_TRIG;
    _p31 : BOOL;
    _p32 : BOOL;
    _p33 : BOOL;
    _e34 : R_TRIG;
END_VAR
(* Network 1 *)
_p1 := gModeControlInterface.Status.BlissPanelAlarmActive;
IF NOT gIO.DIs.SafetyOK OR gServoFeedInterface.Status.Error OR gBodyHopperInterface.Status.Error OR gLeftHopperInterface.Status.Error OR gRightHopperInterface.Status.Error OR gServoRamInterface.Status.Error OR _p1 OR StopFeed OR NOT gServoRamInterface.Status.Homed OR gAlarmActive THEN
    gModeControlInterface.Commands.SetAutoMode := FALSE;
    gModeControlInterface.Commands.SetJogMode := FALSE;
    gHMI.Commands.SelectJogMode := FALSE;
    gHMI.Commands.SelectAutoMode := FALSE;
    gModeControlInterface.Status.Dwelling := FALSE;
END_IF;

(* Network 2 *)
IF NOT gServoRamInterface.Status.Homed THEN gModeControlInterface.Status.Dwelling := FALSE; END_IF;

(* Network 3 *)
IF gHMI.Commands.SelectAutoMode THEN
    gModeControlInterface.Commands.SetAutoMode := TRUE;
    gModeControlInterface.Commands.SetJogMode := FALSE;
END_IF;

(* Network 4 *)
gModeControlInterface.Commands.SetShowMode := gHMI.Commands.EnableShowMode;

(* Network 5 *)
IF gHMI.Commands.SelectJogMode THEN
    gModeControlInterface.Commands.SetJogMode := TRUE;
    gModeControlInterface.Commands.SetAutoMode := FALSE;
    gHMI.Commands.RequestVFDRun := FALSE;
END_IF;

(* Network 6 *)
IF gModeControlInterface.Commands.SetJogMode THEN
    gHMI.ColorMapDatapoints.JogModeSelected := 1;
    gHMI.ColorMapDatapoints.AutoModeSelected := 0;
    gHMI.StatusDatapoints.JogStatusDatapoint := UNHIDE + UNLOCK;
END_IF;

(* Network 7 *)
IF gModeControlInterface.Commands.SetAutoMode THEN
    gHMI.ColorMapDatapoints.JogModeSelected := 0;
    gHMI.ColorMapDatapoints.AutoModeSelected := 1;
    gHMI.StatusDatapoints.JogStatusDatapoint := HIDE + LOCK;
END_IF;

(* Network 8 *)
_p2 := NOT gModeControlInterface.Commands.SetAutoMode AND NOT gModeControlInterface.Commands.SetJogMode;
IF _p2 THEN
    gHMI.ColorMapDatapoints.JogModeSelected := 0;
    gHMI.ColorMapDatapoints.AutoModeSelected := 0;
    gHMI.StatusDatapoints.JogStatusDatapoint := HIDE + LOCK;
END_IF;

(* Network 9 *)
_p3 := gHMI.Commands.SelectAutoMode;
IF _p3 THEN gHMI.StatusDatapoints.AutoModeSDP := UNHIDE + UNLOCK; END_IF;

(* Network 10 *)
_p4 := NOT gHMI.Commands.SelectAutoMode;
IF _p4 THEN gHMI.StatusDatapoints.AutoModeSDP := HIDE + LOCK; END_IF;

(* Network 11: General Lamp Flasher Circuit *)
FlashON(IN := NOT FlashOFF.Q, PT := T#500ms);

(* Network 12: General Lamp Flasher *)
FlashOFF(IN := FlashON.Q, PT := T#500ms);

(* Network 13 *)
gHMI.BitmapSelectDatapoints.ResetPress := (NOT gIO.DIs.SafetyOK AND FlashON.Q) OR gHMI.Commands.RequestReset OR gIO.DIs.SafetyOK;

(* Network 14 *)
gHMI.BitmapSelectDatapoints.StopPress := gHMI.Commands.RequestStop;

(* Network 15 *)
_e5(CLK := gHMI.Commands.RequestStop);
IF NOT gIO.DIs.SafetyOK OR gServoFeedInterface.Status.Error OR gBodyHopperInterface.Status.Error OR gLeftHopperInterface.Status.Error OR gRightHopperInterface.Status.Error OR gServoRamInterface.Status.Error OR gModeControlInterface.Status.BlissPanelAlarmActive OR _e5.Q THEN
    gHMI.Commands.RequestVFDRun := FALSE;
END_IF;

(* Network 16 *)
gHMI.BitmapSelectDatapoints.RunPress := ((gIO.DIs.SafetyOK AND NOT gServoRamInterface.Status.InMotion AND FlashON.Q) OR gModeControlInterface.Status.Dwelling OR gModeControlInterface.Status.WaitingOnDownstream OR gServoFeedInterface.Status.InMotion) AND gHMI.Commands.SelectAutoMode;

(* Network 17 *)
gVacCtrlInterface.Commands.VacuumOn := (gHMI.Commands.RequestVacuumOn OR (NOT gHMI.Commands.RequestVacuumOn AND FlashON.Q)) AND gHMI.Commands.RequestVacuumOn;
gHMI.BitmapSelectDatapoints.VacuumPress := gHMI.Commands.RequestVacuumOn OR (NOT gHMI.Commands.RequestVacuumOn AND FlashON.Q);

(* Network 18 *)
status := SetPatternSDPs(NumGlueChannels := gAdhesiveCtrlInterface.Parameters.NumAdhesiveChannels, FieldColormaps := ADR(gHMI.ColorMapDatapoints), FieldSDPs := ADR(gHMI.StatusDatapoints));

(* Network 19 *)
IF gUserLevel < 1 THEN gHMI.StatusDatapoints.MaintenanceSDP := HIDE + LOCK; END_IF;

(* Network 20 *)
IF gUserLevel > 0 THEN gHMI.StatusDatapoints.MaintenanceSDP := UNHIDE + UNLOCK; END_IF;

(* Network 21 *)
_p6 := NOT gIO.DIs.AdhesiveUnitReady AND gAdhesiveCtrlInterface.Parameters.FeedbackIsHardwire;
_p7 := NOT gAdhesiveCtrlInterface.Parameters.NordsonComms.UnitReady AND gAdhesiveCtrlInterface.Parameters.FeedbackIsModbusTCP;
IF _p6 OR _p7 THEN
    gHMI.StatusDatapoints.AdhesiveUnitNotReadySDP := UNHIDE;
    gHMI.ColorMapDatapoints.AdhesiveUnitReady := NOTOK;
END_IF;

(* Network 22 *)
_p8 := gIO.DIs.AdhesiveUnitReady AND gAdhesiveCtrlInterface.Parameters.FeedbackIsHardwire;
_p9 := gAdhesiveCtrlInterface.Parameters.NordsonComms.UnitReady AND gAdhesiveCtrlInterface.Parameters.FeedbackIsModbusTCP;
IF _p8 OR _p9 THEN
    gHMI.StatusDatapoints.AdhesiveUnitNotReadySDP := HIDE;
    gHMI.ColorMapDatapoints.AdhesiveUnitReady := OK;
END_IF;

(* Network 23 *)
IF NOT gIO.DIs.AdhesiveUnitNotFaulted THEN
    gHMI.StatusDatapoints.AdhesiveUnitFaultSDP := UNHIDE;
    gHMI.ColorMapDatapoints.AdhesiveUnitFault := NOTOK;
END_IF;

(* Network 24 *)
IF gIO.DIs.AdhesiveUnitNotFaulted THEN
    gHMI.StatusDatapoints.AdhesiveUnitFaultSDP := HIDE;
    gHMI.ColorMapDatapoints.AdhesiveUnitFault := OK;
END_IF;

(* Network 25 *)
IF gIO.DIs.AdhesiveLevelLow THEN
    gHMI.StatusDatapoints.AdhesiveUnitLevelLowSDP := UNHIDE;
    gHMI.ColorMapDatapoints.AdhesiveUnitLevelLow := NOTOK;
END_IF;

(* Network 26 *)
IF NOT gIO.DIs.AdhesiveLevelLow THEN
    gHMI.StatusDatapoints.AdhesiveUnitLevelLowSDP := HIDE;
    gHMI.ColorMapDatapoints.AdhesiveUnitLevelLow := OK;
END_IF;

(* Network 27 *)
IF gIO.DIs.LowAdhesiveUseage THEN
    gHMI.StatusDatapoints.AdhesiveUseageLowSDP := UNHIDE;
    gHMI.ColorMapDatapoints.AdhesiveUseageLow := NOTOK;
END_IF;

(* Network 28 *)
IF NOT gIO.DIs.LowAdhesiveUseage THEN
    gHMI.StatusDatapoints.AdhesiveUseageLowSDP := HIDE;
    gHMI.ColorMapDatapoints.AdhesiveUseageLow := OK;
END_IF;

(* Network 29 *)
IF NOT gIO.DIs.VacuumPressureOK THEN gHMI.StatusDatapoints.VacuumPressureFaultSDP := OK; END_IF;

(* Network 30 *)
IF gIO.DIs.VacuumPressureOK THEN gHMI.StatusDatapoints.VacuumPressureFaultSDP := NOTOK; END_IF;

(* Network 31 *)
IF gIO.DOs.VacuumOn THEN gHMI.ColorMapDatapoints.VacuumPumpOn := OK; END_IF;

(* Network 32 *)
IF NOT gIO.DOs.VacuumOn THEN gHMI.ColorMapDatapoints.VacuumPumpOn := NOTOK; END_IF;

(* Network 33: *********************************   RECIPE HANDLING      ****************************************** *)
_e10(CLK := gHMI.Commands.LoadRecipe);
IF _e10.Q THEN gRecipeInterface.Commands.LoadRecipe := TRUE; END_IF;

(* Network 34 *)
_e11(CLK := gHMI.Commands.SaveRecipe);
IF _e11.Q THEN gRecipeInterface.Commands.SaveRecipe := TRUE; END_IF;

(* Network 35 *)
_p12 := gHMI.Commands.RequestBoxType1 AND NOT gHMI.Commands.LoadRecipeType1;
_p13 := gHMI.Commands.RequestBoxType1;
IF _p12 THEN
    gHMI.StatusDatapoints.RecipeDialogSDP.0 := FALSE;
    gHMI.Commands.RequestBoxType2 := FALSE;
END_IF;
_p14 := _p13 AND gHMI.Commands.CancelBoxChange;
IF _p13 AND gHMI.Commands.CancelBoxChange THEN gHMI.Commands.RequestBoxType1 := FALSE; END_IF;
IF _p14 THEN
    gHMI.Commands.CancelBoxChange := FALSE;
    gHMI.StatusDatapoints.RecipeDialogSDP.0 := TRUE;
END_IF;
_p15 := _p13 AND gHMI.Commands.ConfirmBoxChange;
IF _p13 AND gHMI.Commands.ConfirmBoxChange THEN gHMI.Commands.LoadRecipeType1 := TRUE; END_IF;
IF _p15 THEN
    gHMI.Commands.ConfirmBoxChange := FALSE;
    gHMI.Commands.RequestBoxType1 := FALSE;
    gHMI.StatusDatapoints.RecipeDialogSDP.0 := TRUE;
END_IF;

(* Network 36 *)
_p16 := gHMI.Commands.RequestBoxType2 AND NOT gHMI.Commands.LoadRecipeType2;
_p17 := gHMI.Commands.RequestBoxType2;
IF _p16 THEN
    gHMI.StatusDatapoints.RecipeDialogSDP.0 := FALSE;
    gHMI.Commands.RequestBoxType1 := FALSE;
END_IF;
_p18 := _p17 AND gHMI.Commands.CancelBoxChange;
IF _p17 AND gHMI.Commands.CancelBoxChange THEN gHMI.Commands.RequestBoxType2 := FALSE; END_IF;
IF _p18 THEN
    gHMI.Commands.CancelBoxChange := FALSE;
    gHMI.StatusDatapoints.RecipeDialogSDP.0 := TRUE;
END_IF;
_p19 := _p17 AND gHMI.Commands.ConfirmBoxChange;
IF _p17 AND gHMI.Commands.ConfirmBoxChange THEN gHMI.Commands.LoadRecipeType2 := TRUE; END_IF;
IF _p19 THEN
    gHMI.Commands.ConfirmBoxChange := FALSE;
    gHMI.Commands.RequestBoxType2 := FALSE;
    gHMI.StatusDatapoints.RecipeDialogSDP.0 := TRUE;
END_IF;

(* Network 37 *)
_e20(CLK := gHMI.Commands.LoadRecipeType1);
IF _e20.Q THEN
    gRecipeInterface.Commands.LoadRecipe := TRUE;
    gHMI.Commands.LoadRecipeType2 := FALSE;
    gHMI.StatusDatapoints.RecipeReq2SDP.1 := FALSE;
    gHMI.StatusDatapoints.RecipeReq1SDP.1 := TRUE;
    gRecipeInterface.Parameters.RecipeName := TYPE1_RECIPE_NAME;
END_IF;

(* Network 38 *)
_e21(CLK := gHMI.Commands.LoadRecipeType2);
IF _e21.Q THEN
    gRecipeInterface.Commands.LoadRecipe := TRUE;
    gHMI.Commands.LoadRecipeType1 := FALSE;
    gHMI.StatusDatapoints.RecipeReq2SDP.1 := TRUE;
    gHMI.StatusDatapoints.RecipeReq1SDP.1 := FALSE;
    gRecipeInterface.Parameters.RecipeName := TYPE2_RECIPE_NAME;
END_IF;

(* Network 39 *)
gHMI.StatusDatapoints.RecipeIndexSDP := gRecipeInterface.Status.LoadedRecipeIndex;

(* Network 40 *)
_p22 := NOT gHMI.Commands.LoadRecipeType1 AND NOT gHMI.Commands.LoadRecipeType2;
IF _p22 THEN gHMI.Commands.LoadRecipeType1 := gHMI.StatusDatapoints.RecipeIndexSDP = 1; END_IF;

(* Network 41 *)
_p23 := NOT gHMI.Commands.LoadRecipeType1 AND NOT gHMI.Commands.LoadRecipeType2;
IF _p23 THEN gHMI.Commands.LoadRecipeType2 := gHMI.StatusDatapoints.RecipeIndexSDP = 2; END_IF;

(* Network 42 *)
IF gRecipeInterface.Status.Busy THEN gHMI.ColorMapDatapoints.RecipeSystemBusy := OK; END_IF;

(* Network 43 *)
IF NOT gRecipeInterface.Status.Busy THEN gHMI.ColorMapDatapoints.RecipeSystemBusy := NOTOK; END_IF;

(* Network 44 *)
SettingsLoaded := gRecipeInterface.Parameters.RecipeName = gRecipeInterface.Status.LoadedRecipeName;

(* Network 45 *)
IF SettingsLoaded THEN gHMI.ColorMapDatapoints.RecipeLoaded := OK; END_IF;

(* Network 46 *)
IF SettingsLoaded THEN gHMI.ColorMapDatapoints.RecipeLoaded := OK; END_IF;

(* Network 47 *)
IF NOT gAlarmActive THEN gHMI.BitmapSelectDatapoints.AlarmActive := ALARM_INACTIVE; END_IF;

(* Network 48 *)
IF gAlarmActive THEN gHMI.BitmapSelectDatapoints.AlarmActive := ALARM_ACTIVE; END_IF;

(* Network 49 *)
IF NOT gAdhesiveCtrlInterface.Status.AlarmActive THEN
    gHMI.ColorMapDatapoints.AdhesiveSystemOK := OK;
END_IF;

(* Network 50 *)
IF gAdhesiveCtrlInterface.Status.AlarmActive THEN
    gHMI.ColorMapDatapoints.AdhesiveSystemOK := NOTOK;
END_IF;

(* Network 51 *)
IF NOT gAirPressureAlarmActive THEN gHMI.ColorMapDatapoints.AirPressureOK := OK; END_IF;

(* Network 52 *)
IF gAirPressureAlarmActive THEN gHMI.ColorMapDatapoints.AirPressureOK := NOTOK; END_IF;

(* Network 53 *)
IF NOT gVacCtrlInterface.Status.AlarmActive THEN gHMI.ColorMapDatapoints.VacuumOK := OK; END_IF;

(* Network 54 *)
IF gVacCtrlInterface.Status.AlarmActive THEN gHMI.ColorMapDatapoints.VacuumOK := NOTOK; END_IF;

(* Network 55 *)
IF NOT gSafetyNotOKAlarmActive THEN gHMI.ColorMapDatapoints.SafetyOK := OK; END_IF;

(* Network 56 *)
IF gSafetyNotOKAlarmActive THEN gHMI.ColorMapDatapoints.SafetyOK := NOTOK; END_IF;

(* Network 57 *)
IF NOT gServoFeedInterface.Status.Error AND NOT gBodyHopperInterface.Status.Error AND NOT gLeftHopperInterface.Status.Error AND NOT gRightHopperInterface.Status.Error AND NOT gServoRamInterface.Status.Error AND NOT gFoldPushCtrlInterface.Parameters.LinMotBotFolder.Status.Error AND NOT gFoldPushCtrlInterface.Parameters.LinMotTopFolder.Status.Error THEN
    gHMI.ColorMapDatapoints.DriveFaultOK := OK;
END_IF;

(* Network 58 *)
IF gServoFeedInterface.Status.Error OR gBodyHopperInterface.Status.Error OR gLeftHopperInterface.Status.Error OR gRightHopperInterface.Status.Error OR gServoRamInterface.Status.Error OR gFoldPushCtrlInterface.Parameters.LinMotBotFolder.Status.Error OR gFoldPushCtrlInterface.Parameters.LinMotTopFolder.Status.Error THEN
    gHMI.ColorMapDatapoints.DriveFaultOK := NOTOK;
END_IF;

(* Network 59 *)
IF gIO.DIs.DownstreamSensor THEN gHMI.ColorMapDatapoints.DownstreamSensorOK := NOTOK; END_IF;

(* Network 60 *)
IF NOT gIO.DIs.DownstreamSensor THEN gHMI.ColorMapDatapoints.DownstreamSensorOK := OK; END_IF;

(* Network 61 *)
IF NOT gFoldPushCtrlInterface.Status.TopFoldValveStatus THEN
    gHMI.ColorMapDatapoints.Valve1OK := NOTOK;
END_IF;

(* Network 62 *)
IF gFoldPushCtrlInterface.Status.TopFoldValveStatus THEN gHMI.ColorMapDatapoints.Valve1OK := OK; END_IF;

(* Network 63 *)
IF NOT gFoldPushCtrlInterface.Status.BottomFoldValveStatus THEN
    gHMI.ColorMapDatapoints.Valve2OK := NOTOK;
END_IF;

(* Network 64 *)
IF gFoldPushCtrlInterface.Status.BottomFoldValveStatus THEN
    gHMI.ColorMapDatapoints.Valve2OK := OK;
END_IF;

(* Network 65 *)
IF NOT gFoldPushCtrlInterface.Status.CompOnValveStatus THEN
    gHMI.ColorMapDatapoints.Valve3OK := NOTOK;
END_IF;

(* Network 66 *)
IF gFoldPushCtrlInterface.Status.CompOnValveStatus THEN gHMI.ColorMapDatapoints.Valve3OK := OK; END_IF;

(* Network 67 *)
IF NOT gFoldPushCtrlInterface.Status.PushValveStatus THEN
    gHMI.ColorMapDatapoints.Valve4OK := NOTOK;
END_IF;

(* Network 68 *)
IF gFoldPushCtrlInterface.Status.PushValveStatus THEN gHMI.ColorMapDatapoints.Valve4OK := OK; END_IF;

(* Network 69 *)
IF gFoldPushCtrlInterface.Status.HardwireConfig THEN
    gHMI.StatusDatapoints.HardwireValveSDP := UNHIDE + UNLOCK;
END_IF;

(* Network 70 *)
IF gIO.SafetyStatus.SafetyProgramRunning THEN gHMI.StatusDatapoints.SafetyStartingSDP := HIDE; END_IF;

(* Network 71 *)
IF NOT gIO.SafetyStatus.SafetyProgramRunning THEN
    gHMI.StatusDatapoints.SafetyStartingSDP := UNHIDE;
END_IF;

(* Network 72 *)
_e24(CLK := gAlarmActive);
IF _e24.Q THEN gChangePage := PAGE_ALARM; END_IF;

(* Network 73 *)
IF gModeControlInterface.Parameters.MachineType = MACHINE_TYPE_BLISS THEN
    gHMI.StatusDatapoints.BlissSDP := UNHIDE + UNLOCK;
END_IF;

(* Network 74 *)
IF gModeControlInterface.Parameters.MachineType <> MACHINE_TYPE_BLISS THEN
    gHMI.StatusDatapoints.BlissSDP := HIDE + LOCK;
END_IF;

(* Network 75 *)
_t25 := gModeControlInterface.Parameters.MachineType = MACHINE_TYPE_CLASSICPAK;
IF _t25 THEN
    gModeControlInterface.Parameters.MaxPPM := 20;
    gModeControlInterface.Parameters.MinPPM := 0;
END_IF;

(* Network 76 *)
_t26 := gModeControlInterface.Parameters.MachineType = MACHINE_TYPE_BLISS;
IF _t26 THEN
    gModeControlInterface.Parameters.MaxPPM := 25;
    gModeControlInterface.Parameters.MinPPM := 0;
END_IF;

(* Network 77 *)
_t27 := gModeControlInterface.Parameters.MachineType = MACHINE_TYPE_TRAY;
IF _t27 THEN
    gModeControlInterface.Parameters.MaxPPM := 25;
    gModeControlInterface.Parameters.MinPPM := 0;
    gHMI.StatusDatapoints.TraySDP := UNHIDE + UNLOCK;
END_IF;

(* Network 78 *)
IF gModeControlInterface.Parameters.MachineType <> MACHINE_TYPE_TRAY THEN
    gHMI.StatusDatapoints.TraySDP := HIDE + LOCK;
END_IF;

(* Network 79 *)
_p28 := gModeControlInterface.Parameters.MaxPPM < gModeControlInterface.Parameters.PiecesPerMinute;
IF _p28 THEN
    gModeControlInterface.Parameters.PiecesPerMinute := gModeControlInterface.Parameters.MaxPPM;
END_IF;

(* Network 80 *)
_p29 := gModeControlInterface.Parameters.MinPPM > gModeControlInterface.Parameters.PiecesPerMinute;
IF _p29 THEN
    gModeControlInterface.Parameters.PiecesPerMinute := gModeControlInterface.Parameters.MinPPM;
END_IF;

(* Network 81 *)
LogoutTimer(IN := NOT ResetTimeoutTimer, PT := T#120s);
ResetUserLevel := LogoutTimer.Q;

(* Network 82 *)
_e30(CLK := ResetUserLevel);
IF _e30.Q THEN
    gUserLevel := 0;
    gChangePage := 0;
END_IF;

(* Network 83 *)
ResetTimeoutTimer := gActivePage <> OldPage;

(* Network 84 *)
OldPage := gActivePage;

(* Network 85 *)
gHMI.StatusDatapoints.LinMotSDP.0 := NOT gFoldPushCtrlInterface.Status.LinMotConfig;
gHMI.StatusDatapoints.LinMotTopHomeSDP.0 := NOT gFoldPushCtrlInterface.Status.LinMotConfig;
gHMI.StatusDatapoints.LinMotBotHomeSDP.0 := NOT gFoldPushCtrlInterface.Status.LinMotConfig;

(* Network 86 *)
_p31 := gHMI.ColorMapDatapoints.AutoModeSelected.0;
gHMI.StatusDatapoints.LinMotTopHomeSDP.1 := gHMI.ColorMapDatapoints.AutoModeSelected.0;
gHMI.StatusDatapoints.LinMotBotHomeSDP.1 := _p31;

(* Network 87 *)
gHMI.StatusDatapoints.PnuematicFolderSDP.0 := NOT gFoldPushCtrlInterface.Status.PneumaticConfig;

(* Network 88 *)
IF gAdhesiveCtrlInterface.Status.ATS_AddOnOverLimit THEN
    gHMI.ColorMapDatapoints.ATSAddOnOver := NOTOK;
END_IF;

(* Network 89 *)
IF NOT gAdhesiveCtrlInterface.Status.ATS_AddOnOverLimit THEN
    gHMI.ColorMapDatapoints.ATSAddOnOver := OK;
END_IF;

(* Network 90 *)
IF gAdhesiveCtrlInterface.Status.ATS_AddOnUnderLimit THEN
    gHMI.ColorMapDatapoints.ATSAddOnUnder := NOTOK;
END_IF;

(* Network 91 *)
IF NOT gAdhesiveCtrlInterface.Status.ATS_AddOnUnderLimit THEN
    gHMI.ColorMapDatapoints.ATSAddOnUnder := OK;
END_IF;

(* Network 92 *)
gAdhesiveCtrlInterface.Parameters.NordsonComms.ChannelDataSize := SIZEOF(in := gAdhesiveCtrlInterface.Parameters.NordsonComms.ChannelSetTempActual);

(* Network 93: Flash save set temp button if  requested temps are different from current set temps *)
gAdhesiveCtrlInterface.Parameters.NordsonComms.ChannelDataCmpResult := brsmemcmp(pMem1 := ADR(gAdhesiveCtrlInterface.Parameters.NordsonComms.ChannelSetTempActual), pMem2 := ADR(gAdhesiveCtrlInterface.Parameters.NordsonComms.ChannelSetTempRequested), length := gAdhesiveCtrlInterface.Parameters.NordsonComms.ChannelDataSize);

(* Network 94 *)
gHMI.ColorMapDatapoints.NordsonEditTemps := gAdhesiveCtrlInterface.Parameters.NordsonComms.ChannelDataCmpResult <> 0;

(* Network 95 *)
gHMI.ColorMapDatapoints.NordsonEditTemps.0 := gHMI.ColorMapDatapoints.NordsonEditTemps.0 AND FlashON.Q;

(* Network 96 *)
IF gIO.DIs.BodyHopperLow OR gIO.DIs.LeftHopperLow OR gIO.DIs.RightHopperLow THEN
    gHMI.StatusDatapoints.HopperLowSDP := UNHIDE + UNLOCK;
END_IF;

(* Network 97 *)
IF NOT gIO.DIs.BodyHopperLow OR NOT gIO.DIs.LeftHopperLow OR NOT gIO.DIs.RightHopperLow THEN
    gHMI.StatusDatapoints.HopperLowSDP := HIDE + LOCK;
END_IF;

(* Network 98 *)
_p32 := NOT gHMI.Commands.CycleServoRam;
IF _p32 THEN gHMI.StatusDatapoints.HomeServoRamSDP := UNHIDE + UNLOCK; END_IF;

(* Network 99 *)
_p33 := gHMI.Commands.CycleServoRam;
IF _p33 THEN gHMI.StatusDatapoints.HomeServoRamSDP := HIDE + LOCK; END_IF;

(* Network 100 *)
IF LubricationOK THEN gHMI.StatusDatapoints.LubeSDP := HIDE + LOCK; END_IF;

(* Network 101 *)
IF NOT LubricationOK THEN gHMI.StatusDatapoints.LubeSDP := UNHIDE + UNLOCK; END_IF;

(* Network 102 *)
_e34(CLK := gHMI.StatusDatapoints.AdhesivePatternConfirmedSDP.0);
IF _e34.Q THEN
    gHMI.StatusDatapoints.AdhesivePatternConfirmDialogSDP.0 := TRUE;
    gHMI.StatusDatapoints.AdhesivePatternDialogSDP.0 := TRUE;
END_IF;

(* Network 103: Controls whether or not the text is shown on screen for the respective hopper switches being off. Setting the first bit true hides the text *)
gHMI.StatusDatapoints.BodyHopperSwitchSDP.0 := gIO.DIs.BodyHopperMotor_RUN;

(* Network 104 *)
gHMI.StatusDatapoints.LeftHopperSwitchSDP.0 := gIO.DIs.LeftHopperMotor_RUN;

(* Network 105 *)
gHMI.StatusDatapoints.RightHopperSwitchSDP.0 := gIO.DIs.RightHopperMotor_RUN;
END_PROGRAM
```

- Visualisation Logical/HMI/Visu (not shown)

- Visualisation Logical/HMI/Visu_Resized (not shown)

### Program Logical/ModeControl/ModeControl

#### Init.st
```iecst
PROGRAM _INIT

	//asign default values to parameters
	//defaults, not needed
	(*
	gModeControlInterface.Parameters.PiecesPerMinute := 10;
	gModeControlInterface.Parameters.DwellTime := 0; //ms
	gModeControlInterface.Parameters.StopPosition := 0;

	gAdhesiveCtrlInterface.Parameters.AdhesivePatterns[0].DelayDistance[0] := 150;
	gAdhesiveCtrlInterface.Parameters.AdhesivePatterns[1].DelayDistance[0] := 150;
	gAdhesiveCtrlInterface.Parameters.AdhesivePatterns[2].DelayDistance[0] := 150;
	gAdhesiveCtrlInterface.Parameters.AdhesivePatterns[3].DelayDistance[0] := 150;

	gAdhesiveCtrlInterface.Parameters.AdhesivePatterns[0].GlueOnDistance[0] := 32;
	gAdhesiveCtrlInterface.Parameters.AdhesivePatterns[1].GlueOnDistance[0] := 32;
	gAdhesiveCtrlInterface.Parameters.AdhesivePatterns[2].GlueOnDistance[0] := 32;
	gAdhesiveCtrlInterface.Parameters.AdhesivePatterns[3].GlueOnDistance[0] := 32;

	gAdhesiveCtrlInterface.Parameters.AdhesivePatterns[0].DelayDistance[1] := 210;
	gAdhesiveCtrlInterface.Parameters.AdhesivePatterns[1].DelayDistance[1] := 210;
	gAdhesiveCtrlInterface.Parameters.AdhesivePatterns[2].DelayDistance[1] := 210;
	gAdhesiveCtrlInterface.Parameters.AdhesivePatterns[3].DelayDistance[1] := 210;

	gAdhesiveCtrlInterface.Parameters.AdhesivePatterns[0].GlueOnDistance[1] := 32;
	gAdhesiveCtrlInterface.Parameters.AdhesivePatterns[1].GlueOnDistance[1] := 32;
	gAdhesiveCtrlInterface.Parameters.AdhesivePatterns[2].GlueOnDistance[1] := 32;
	gAdhesiveCtrlInterface.Parameters.AdhesivePatterns[3].GlueOnDistance[1] := 32;

	gAdhesiveCtrlInterface.Parameters.AdhesivePatterns[0].DelayDistance[2] := 300;
	gAdhesiveCtrlInterface.Parameters.AdhesivePatterns[1].DelayDistance[2] := 300;
	gAdhesiveCtrlInterface.Parameters.AdhesivePatterns[2].DelayDistance[2] := 300;
	gAdhesiveCtrlInterface.Parameters.AdhesivePatterns[3].DelayDistance[2] := 300;

	gAdhesiveCtrlInterface.Parameters.AdhesivePatterns[0].GlueOnDistance[2] := 32;
	gAdhesiveCtrlInterface.Parameters.AdhesivePatterns[1].GlueOnDistance[2] := 32;
	gAdhesiveCtrlInterface.Parameters.AdhesivePatterns[2].GlueOnDistance[2] := 32;
	gAdhesiveCtrlInterface.Parameters.AdhesivePatterns[3].GlueOnDistance[2] := 32;

	gFoldPushCtrlInterface.Parameters.BottomFolderOnPos := 100;
	gFoldPushCtrlInterface.Parameters.BottomFolderOffPos := 200;
	gFoldPushCtrlInterface.Parameters.TopFolderOnPos := 180;
	gFoldPushCtrlInterface.Parameters.TopFolderOffPos := 300;
	*)

	gPassword;
	gUserLevel;
	gIO;

	//set these DI's true. physical IO will take over once program runs,
	//and we need to make sure we see a falling edge on these IO points so that alarms are reported
	gIO.DIs.SafetyOK := TRUE;
	gIO.SafetyStatus.BackEstopOK := TRUE;
	gIO.SafetyStatus.FrontEStopOK := TRUE;
	gIO.SafetyStatus.GuardDoorsOK := TRUE;
	gIO.DIs.AirPressureOK := TRUE;
	gIO.DIs.VacuumPressureOK := TRUE;
	gIO.DIs.AdhesiveUnitNotFaulted := TRUE;
	gIO.DIs.AdhesiveUnitReady := TRUE;
	gIO.DIs.AdhesiveLevelLow := FALSE;
	gIO.DIs.VacuumTempOK := TRUE;
	gIO.DIs.BodyHopperLow := TRUE;

	gAutoTune := FALSE;
	gCurrentLimitHit := FALSE;

	//PickDwellTime := T#
	gHMI.Parameters.PickDwellTime :=0;
	gHMI.Parameters.PickAndPlaceDwell := 750; //750 ms
	gHMI.Parameters.LowHopperTime := 3000; //3S
	gHMI.Parameters.LowFeedJamTime := 10000; // 3S
	gHMI.Parameters.TopFeedJamTime := 10000; // 3 S
	gHMI.Parameters.VacuumOffTime := 1000; // 1 S
	gHMI.Parameters.DownPulseTime := 1000; // 1 S
	gHMI.Parameters.Y_DelayTime := 500; // 500ms
	gHMI.Parameters.BlowOffTime := 10; // 10ms
	gHMI.Parameters.LubeCycleCount := 5; // 5 cycles
	gHMI.Parameters.SetCycleCount := 25000; // 25000 Ram Servo Cycles

END_PROGRAM
```

### Program Logical/ModeControl/ModeControl_ST

#### Variables.var
```iecst
VAR
	AirPressureAlarmActive : BOOL;
	AirPressureNotOK : BOOL;
	AirPressureNotOKTimer : TON;
	BlowOff_Pulse : TP;
	BlowOff_Trigger : BOOL;
	PnPTimeoutError : BOOL;
	BodyCheckError : BOOL;
	InfeedCheckError : BOOL;
	BodyCheckErrorActive : BOOL;
	BodyHopperLowAlarm : BOOL;
	BodyHopperLowTMR : TON;
	BodyPanelTimeout : TON;
	InfeedTimeout : TON;
	BoxPickTMR : TON;
	CountReset : BOOL;
	DistanceFromStopPosition : REAL;
	DownstreamBlocked : BOOL;
	DownstreamSensorONTimer : TON;
	DownstreamSensorTimer : TON;
	Dummy : BOOL;
	DwellTimer : TON;
	EuchnerSafeResetTimer : TON;
	FeedPosFinal : LREAL;
	FeedPositionCapture : LREAL;
	FeedServoPosSP : LREAL;
	FeedServoTimeout : BOOL;
	FeedServoTMR : TON;
	FeedStopTimer : TON;
	ForceBodyPanellError : BOOL;
	FrontEStopNotOKActive : BOOL;
END_VAR
VAR CONSTANT
	Ftrig_BlowOffOnManual : F_TRIG := (0); (*Falling edge detection function block for this variable*)
END_VAR
VAR
	Ftrig_DownstreamBlocked : F_TRIG;
	GluePhotoEyeAlarmActive : BOOL;
	GuardDoorNotOKActive : BOOL;
	HopperRunningError : BOOL;
	InBlissSidePanelCheckWindow : BOOL;
	LeftHopperLowAlarm : BOOL;
	LeftHopperLowTMR : TON;
	LubeReset : BOOL;
	LubricationCounter : CTU;
	MoveVelocityRequest : BOOL;
	PnPTimeout : TON;
	OldEncoderPos : REAL;
	PhotoEyeCheckErrorActive : BOOL;
	PhotoEyeTimeout : TON;
	PickAndPlaceDwelling : BOOL;
	PickAndPlaceDwellTimer : TON;
	PickAndPlaceHasBox : BOOL;
	PickDwellTime : TIME;
	RamAtStopPosition : BOOL;
	RamCycleCount : UDINT;
	RearEStopNotOKActive : BOOL;
	Return_Trigger : BOOL;
	RightHopperLowAlarm : BOOL;
	RightHopperLowTMR : TON;
	Rtrig_AlarmActive : R_TRIG; (*Rising edge detection function block for this variable*)
	Rtrig_BlowOffManual : R_TRIG; (*Rising edge detection function block for this variable*)
	Rtrig_BlowOffTrigger : R_TRIG; (*Rising edge detection function block for this variable*)
	Rtrig_DownstreamBlocked : R_TRIG; (*Rising edge detection function block for this variable*)
	Rtrig_FeedServoTMR : R_TRIG; (*Rising edge detection function block for this variable*)
	Rtrig_HopperLow : R_TRIG; (*Rising edge detection function block for this variable*)
	Rtrig_InfeedBoxPresent : R_TRIG; (*Rising edge detection function block for this variable*)
	Rtrig_LubricationCounter : R_TRIG; (*Rising edge detection function block for this variable*)
	Rtrig_PhotoEyeSeen : R_TRIG; (*Rising edge detection function block for this variable*)
	Rtrig_RequestStop : R_TRIG; (*Rising edge detection function block for this variable*)
	Rtrig_RequestVFDRun : R_TRIG;
	SafetyNotOKActive : BOOL;
	SafetyResetRequestTimer : TON;
	ShowModeTimer : TON;
	SideCheckError : BOOL;
	SideCheckErrorActive : BOOL;
	status : UDINT;
	StopFeedServo : BOOL;
	StopPositionDwellExpire : BOOL;
	StopTriggerByDownstream : BOOL;
	TON_BlowOff : TON; (*Timer for blow off after vacuum is shut off (user defined time)*)
	TON_RamDelay : TON; (*Timer for the Ram to delay forward motion*)
	VaccumStopTimer : TON;
	VacuumOffTime : TIME;
	VacuumTimer : TON;
	Vacuum_ON : BOOL;
	Y_Delay : TON;
	Y_Down_Pulse : TP;
	Y_Trigger : BOOL;
END_VAR
```
